   DATA[726,15] := 1.0;
   DATA[726,16] := 1.0;
   DATA[726,17] := 1.0;
   DATA[726,18] := 1.0;
   DATA[726,19] := 1.0;
   DATA[726,20] := 148.808;
   DATA[726,21] := 155.8318;
   DATA[726,22] := 1.720309;
   DATA[726,23] := 999.9744;
   DATA[726,24] := 2.0;
   DATA[726,25] := 2.0;
   DATA[726,26] := 7.878942;
   DATA[726,27] := 144.6039;
   DATA[726,28] := 263.1056;
   DATA[726,29] := 12.11228;
   DATA[726,30] := 1.734683;
   DATA[726,31] := 1.301652;
   DATA[726,32] := 0.7352687;
   DATA[726,33] := 0.3066329;
   DATA[726,34] := 2.0;
   DATA[726,35] := 251.474;
   DATA[726,36] := 1.730048;
   DATA[726,37] := 190.1275;
   DATA[726,38] := 0.000128152;
   DATA[726,39] := 1.0;
   DATA[727,0] := 2.455241;
   DATA[727,1] := 535.5254;
   DATA[727,2] := 2.0;
   DATA[727,3] := 2.0;
   DATA[727,4] := 262.1764;
   DATA[727,5] := 8.395475;
   DATA[727,6] := 327.6339;
   DATA[727,7] := 2.440393;
   DATA[727,8] := 2.0;
   DATA[727,9] := 2.0;
   DATA[727,10] := 2.0;
   DATA[727,11] := 1.987963;
   DATA[727,13] := 991.052;
   DATA[727,14] := 1.0;
   DATA[727,15] := 1.0;
   DATA[727,16] := 1.0;
   DATA[727,17] := 1.0;
   DATA[727,18] := 1.0;
   DATA[727,19] := 1.0;
   DATA[727,20] := 148.808;
   DATA[727,21] := 155.8318;
   DATA[727,22] := 1.720309;
   DATA[727,23] := 1000.051;
   DATA[727,24] := 2.0;
   DATA[727,25] := 2.0;
   DATA[727,26] := 7.878942;
   DATA[727,27] := 144.6039;
   DATA[727,28] := 263.1056;
   DATA[727,29] := 12.11228;
   DATA[727,30] := 1.734683;
   DATA[727,31] := 1.301652;
   DATA[727,32] := 0.7352687;
   DATA[727,33] := 0.3066329;
   DATA[727,34] := 2.0;
   DATA[727,35] := 251.474;
   DATA[727,36] := 1.730048;
   DATA[727,37] := 190.1275;
   DATA[727,38] := 0.000128152;
   DATA[727,39] := 1.0;
   DATA[728,0] := 2.444031;
   DATA[728,1] := 535.4076;
   DATA[728,2] := 2.0;
   DATA[728,3] := 2.0;
   DATA[728,4] := 262.1764;
   DATA[728,5] := 8.395475;
   DATA[728,6] := 327.6339;
   DATA[728,7] := 2.440393;
   DATA[728,8] := 2.0;
   DATA[728,9] := 2.0;
   DATA[728,10] := 2.0;
   DATA[728,11] := 1.987963;
   DATA[728,13] := 991.2122;
   DATA[728,14] := 1.0;
   DATA[728,15] := 1.0;
   DATA[728,16] := 1.0;
   DATA[728,17] := 1.0;
   DATA[728,18] := 1.0;
   DATA[728,19] := 1.0;
   DATA[728,20] := 148.808;
   DATA[728,21] := 155.8062;
   DATA[728,22] := 1.722231;
   DATA[728,23] := 999.8975;
   DATA[728,24] := 2.0;
   DATA[728,25] := 2.0;
   DATA[728,26] := 7.878942;
   DATA[728,27] := 144.5783;
   DATA[728,28] := 263.1056;
   DATA[728,29] := 12.11228;
   DATA[728,30] := 1.73212;
   DATA[728,31] := 1.292046;
   DATA[728,32] := 0.7352687;
   DATA[728,33] := 0.3066329;
   DATA[728,34] := 2.0;
   DATA[728,35] := 251.474;
   DATA[728,36] := 1.730048;
   DATA[728,37] := 190.1275;
   DATA[728,38] := 0.000128152;
   DATA[728,39] := 1.0;
   DATA[729,0] := 2.43026;
   DATA[729,1] := 535.3291;
   DATA[729,2] := 2.0;
   DATA[729,3] := 2.0;
   DATA[729,4] := 262.1764;
   DATA[729,5] := 8.395475;
   DATA[729,6] := 327.5827;
   DATA[729,7] := 2.440393;
   DATA[729,8] := 2.0;
   DATA[729,9] := 2.0;
   DATA[729,10] := 2.0;
   DATA[729,11] := 2.016774;
   DATA[729,13] := 991.5327;
   DATA[729,14] := 1.0;
   DATA[729,15] := 1.0;
   DATA[729,16] := 1.0;
   DATA[729,17] := 1.0;
   DATA[729,18] := 1.0;
   DATA[729,19] := 1.0;
   DATA[729,20] := 148.808;
   DATA[729,21] := 155.8062;
   DATA[729,22] := 1.722231;
   DATA[729,23] := 999.859;
   DATA[729,24] := 2.0;
   DATA[729,25] := 2.0;
   DATA[729,26] := 7.878942;
   DATA[729,27] := 144.5783;
   DATA[729,28] := 263.1056;
   DATA[729,29] := 12.11228;
   DATA[729,30] := 1.73212;
   DATA[729,31] := 1.292046;
   DATA[729,32] := 0.7352687;
   DATA[729,33] := 0.3066329;
   DATA[729,34] := 2.0;
   DATA[729,35] := 251.474;
   DATA[729,36] := 1.730048;
   DATA[729,37] := 190.1275;
   DATA[729,38] := 0.000128152;
   DATA[729,39] := 1.0;
   DATA[730,0] := 2.424815;
   DATA[730,1] := 535.4076;
   DATA[730,2] := 2.0;
   DATA[730,3] := 2.0;
   DATA[730,4] := 262.1764;
   DATA[730,5] := 8.395475;
   DATA[730,6] := 327.5827;
   DATA[730,7] := 2.440393;
   DATA[730,8] := 2.0;
   DATA[730,9] := 2.0;
   DATA[730,10] := 2.0;
   DATA[730,11] := 2.016774;
   DATA[730,13] := 991.6528;
   DATA[730,14] := 1.0;
   DATA[730,15] := 1.0;
   DATA[730,16] := 1.0;
   DATA[730,17] := 1.0;
   DATA[730,18] := 1.0;
   DATA[730,19] := 1.0;
   DATA[730,20] := 148.808;
   DATA[730,21] := 155.8062;
   DATA[730,22] := 1.722231;
   DATA[730,23] := 999.2822;
   DATA[730,24] := 2.0;
   DATA[730,25] := 2.0;
   DATA[730,26] := 7.878942;
   DATA[730,27] := 144.5783;
   DATA[730,28] := 263.1056;
   DATA[730,29] := 12.11228;
   DATA[730,30] := 1.73212;
   DATA[730,31] := 1.285513;
   DATA[730,32] := 0.7352687;
   DATA[730,33] := 0.3066329;
   DATA[730,34] := 2.0;
   DATA[730,35] := 251.474;
   DATA[730,36] := 1.730048;
   DATA[730,37] := 190.1275;
   DATA[730,38] := 0.000128152;
   DATA[730,39] := 1.0;
   DATA[731,0] := 2.424815;
   DATA[731,1] := 535.4861;
   DATA[731,2] := 2.0;
   DATA[731,3] := 2.0;
   DATA[731,4] := 262.1764;
   DATA[731,5] := 8.395475;
   DATA[731,6] := 327.5827;
   DATA[731,7] := 2.440393;
   DATA[731,8] := 2.0;
   DATA[731,9] := 2.0;
   DATA[731,10] := 2.0;
   DATA[731,11] := 2.016774;
   DATA[731,13] := 992.2136;
   DATA[731,14] := 1.0;
   DATA[731,15] := 1.0;
   DATA[731,16] := 1.0;
   DATA[731,17] := 1.0;
   DATA[731,18] := 1.0;
   DATA[731,19] := 1.0;
   DATA[731,20] := 148.808;
   DATA[731,21] := 155.8062;
   DATA[731,22] := 1.720053;
   DATA[731,23] := 999.2438;
   DATA[731,24] := 2.0;
   DATA[731,25] := 2.0;
   DATA[731,26] := 7.878942;
   DATA[731,27] := 144.5783;
   DATA[731,28] := 263.1056;
   DATA[731,29] := 12.11228;
   DATA[731,30] := 1.730838;
   DATA[731,31] := 1.274497;
   DATA[731,32] := 0.7352687;
   DATA[731,33] := 0.3066329;
   DATA[731,34] := 2.0;
   DATA[731,35] := 251.3939;
   DATA[731,36] := 1.730048;
   DATA[731,37] := 190.1275;
   DATA[731,38] := 0.000128152;
   DATA[731,39] := 1.0;
   DATA[732,0] := 2.452359;
   DATA[732,1] := 535.8002;
   DATA[732,2] := 2.0;
   DATA[732,3] := 2.0;
   DATA[732,4] := 262.1764;
   DATA[732,5] := 8.395475;
   DATA[732,6] := 327.5827;
   DATA[732,7] := 2.440393;
   DATA[732,8] := 2.0;
   DATA[732,9] := 2.0;
   DATA[732,10] := 2.0;
   DATA[732,11] := 2.016774;
   DATA[732,13] := 992.6942;
   DATA[732,14] := 1.0;
   DATA[732,15] := 1.0;
   DATA[732,16] := 1.0;
   DATA[732,17] := 1.0;
   DATA[732,18] := 1.0;
   DATA[732,19] := 1.0;
   DATA[732,20] := 148.808;
   DATA[732,21] := 155.8062;
   DATA[732,22] := 1.720053;
   DATA[732,23] := 998.4747;
   DATA[732,24] := 2.0;
   DATA[732,25] := 2.0;
   DATA[732,26] := 7.878942;
   DATA[732,27] := 144.5783;
   DATA[732,28] := 263.1056;
   DATA[732,29] := 12.11228;
   DATA[732,30] := 1.730838;
   DATA[732,31] := 1.280517;
   DATA[732,32] := 0.7352687;
   DATA[732,33] := 0.3066329;
   DATA[732,34] := 2.0;
   DATA[732,35] := 251.2977;
   DATA[732,36] := 1.730048;
   DATA[732,37] := 190.0154;
   DATA[732,38] := 0.000128152;
   DATA[732,39] := 1.0;
   DATA[733,0] := 2.48887;
   DATA[733,1] := 535.9179;
   DATA[733,2] := 2.0;
   DATA[733,3] := 2.0;
   DATA[733,4] := 262.1764;
   DATA[733,5] := 8.395475;
   DATA[733,6] := 327.5827;
   DATA[733,7] := 2.440393;
   DATA[733,8] := 2.0;
   DATA[733,9] := 2.0;
   DATA[733,10] := 2.0;
   DATA[733,11] := 2.010372;
   DATA[733,13] := 993.4552;
   DATA[733,14] := 1.0;
   DATA[733,15] := 1.0;
   DATA[733,16] := 1.0;
   DATA[733,17] := 1.0;
   DATA[733,18] := 1.0;
   DATA[733,19] := 1.0;
   DATA[733,20] := 148.808;
   DATA[733,21] := 155.8062;
   DATA[733,22] := 1.720053;
   DATA[733,23] := 998.6285;
   DATA[733,24] := 2.0;
   DATA[733,25] := 2.0;
   DATA[733,26] := 7.878942;
   DATA[733,27] := 144.5783;
   DATA[733,28] := 263.1056;
   DATA[733,29] := 12.11228;
   DATA[733,30] := 1.730838;
   DATA[733,31] := 1.28167;
   DATA[733,32] := 0.7352687;
   DATA[733,33] := 0.3066329;
   DATA[733,34] := 2.0;
   DATA[733,35] := 251.2977;
   DATA[733,36] := 1.730048;
   DATA[733,37] := 190.0154;
   DATA[733,38] := 0.000128152;
   DATA[733,39] := 1.0;
   DATA[734,0] := 2.532428;
   DATA[734,1] := 535.4076;
   DATA[734,2] := 2.0;
   DATA[734,3] := 2.0;
   DATA[734,4] := 262.1764;
   DATA[734,5] := 8.395475;
   DATA[734,6] := 327.5827;
   DATA[734,7] := 2.440393;
   DATA[734,8] := 2.0;
   DATA[734,9] := 2.0;
   DATA[734,10] := 2.0;
   DATA[734,11] := 2.003969;
   DATA[734,13] := 993.6956;
   DATA[734,14] := 1.0;
   DATA[734,15] := 1.0;
   DATA[734,16] := 1.0;
   DATA[734,17] := 1.0;
   DATA[734,18] := 1.0;
   DATA[734,19] := 1.0;
   DATA[734,20] := 148.808;
   DATA[734,21] := 155.8062;
   DATA[734,22] := 1.720053;
   DATA[734,23] := 998.1287;
   DATA[734,24] := 2.0;
   DATA[734,25] := 2.0;
   DATA[734,26] := 7.878942;
   DATA[734,27] := 144.7321;
   DATA[734,28] := 263.1056;
   DATA[734,29] := 12.11228;
   DATA[734,30] := 1.730838;
   DATA[734,31] := 1.296273;
   DATA[734,32] := 0.7352687;
   DATA[734,33] := 0.3066329;
   DATA[734,34] := 2.0;
   DATA[734,35] := 251.2977;
   DATA[734,36] := 1.730048;
   DATA[734,37] := 190.0154;
   DATA[734,38] := 0.000128152;
   DATA[734,39] := 1.0;
   DATA[735,0] := 2.572783;
   DATA[735,1] := 534.9366;
   DATA[735,2] := 2.0;
   DATA[735,3] := 2.0;
   DATA[735,4] := 262.1764;
   DATA[735,5] := 8.395475;
   DATA[735,6] := 327.5827;
   DATA[735,7] := 2.440393;
   DATA[735,8] := 2.0;
   DATA[735,9] := 2.0;
   DATA[735,10] := 2.0;
   DATA[735,11] := 2.003969;
   DATA[735,13] := 994.4165;
   DATA[735,14] := 1.0;
   DATA[735,15] := 1.0;
   DATA[735,16] := 1.0;
   DATA[735,17] := 1.0;
   DATA[735,18] := 1.0;
   DATA[735,19] := 1.0;
   DATA[735,20] := 148.808;
   DATA[735,21] := 155.8062;
   DATA[735,22] := 1.720053;
   DATA[735,23] := 998.244;
   DATA[735,24] := 2.0;
   DATA[735,25] := 2.0;
   DATA[735,26] := 7.878942;
   DATA[735,27] := 144.7321;
   DATA[735,28] := 263.1056;
   DATA[735,29] := 12.11228;
   DATA[735,30] := 1.730838;
   DATA[735,31] := 1.299475;
   DATA[735,32] := 0.7352687;
   DATA[735,33] := 0.3066329;
   DATA[735,34] := 2.0;
   DATA[735,35] := 251.2977;
   DATA[735,36] := 1.730048;
   DATA[735,37] := 189.9994;
   DATA[735,38] := 0.000128152;
   DATA[735,39] := 1.0;
   DATA[736,0] := 2.609615;
   DATA[736,1] := 534.8581;
   DATA[736,2] := 2.0;
   DATA[736,3] := 2.0;
   DATA[736,4] := 262.1764;
   DATA[736,5] := 8.395475;
   DATA[736,6] := 327.5827;
   DATA[736,7] := 2.440393;
   DATA[736,8] := 2.0;
   DATA[736,9] := 2.0;
   DATA[736,10] := 2.0;
   DATA[736,11] := 2.003969;
   DATA[736,13] := 994.8972;
   DATA[736,14] := 1.0;
   DATA[736,15] := 1.0;
   DATA[736,16] := 1.0;
   DATA[736,17] := 1.0;
   DATA[736,18] := 1.0;
   DATA[736,19] := 1.0;
   DATA[736,20] := 148.808;
   DATA[736,21] := 155.8062;
   DATA[736,22] := 1.720053;
   DATA[736,23] := 997.8979;
   DATA[736,24] := 2.0;
   DATA[736,25] := 2.0;
   DATA[736,26] := 7.878942;
   DATA[736,27] := 144.7321;
   DATA[736,28] := 263.1056;
   DATA[736,29] := 12.11228;
   DATA[736,30] := 1.730838;
   DATA[736,31] := 1.292046;
   DATA[736,32] := 0.7352687;
   DATA[736,33] := 0.3066329;
   DATA[736,34] := 2.0;
   DATA[736,35] := 251.2977;
   DATA[736,36] := 1.730048;
   DATA[736,37] := 189.9994;
   DATA[736,38] := 0.000128152;
   DATA[736,39] := 1.0;
   DATA[737,0] := 2.633635;
   DATA[737,1] := 534.5048;
   DATA[737,2] := 2.0;
   DATA[737,3] := 2.0;
   DATA[737,4] := 262.1764;
   DATA[737,5] := 8.395475;
   DATA[737,6] := 327.5827;
   DATA[737,7] := 2.440393;
   DATA[737,8] := 2.0;
   DATA[737,9] := 2.0;
   DATA[737,10] := 2.0;
   DATA[737,11] := 2.003969;
   DATA[737,13] := 995.4178;
   DATA[737,14] := 1.0;
   DATA[737,15] := 1.0;
   DATA[737,16] := 1.0;
   DATA[737,17] := 1.0;
   DATA[737,18] := 1.0;
   DATA[737,19] := 1.0;
   DATA[737,20] := 148.808;
   DATA[737,21] := 155.8062;
   DATA[737,22] := 1.720053;
   DATA[737,23] := 997.475;
   DATA[737,24] := 2.0;
   DATA[737,25] := 2.0;
   DATA[737,26] := 7.878942;
   DATA[737,27] := 144.7321;
   DATA[737,28] := 263.1056;
   DATA[737,29] := 12.11228;
   DATA[737,30] := 1.730838;
   DATA[737,31] := 1.28167;
   DATA[737,32] := 0.7352687;
   DATA[737,33] := 0.3066329;
   DATA[737,34] := 2.0;
   DATA[737,35] := 251.2977;
   DATA[737,36] := 1.730048;
   DATA[737,37] := 189.9994;
   DATA[737,38] := 0.000128152;
   DATA[737,39] := 1.0;
   DATA[738,0] := 2.649649;
   DATA[738,1] := 534.3085;
   DATA[738,2] := 2.0;
   DATA[738,3] := 2.0;
   DATA[738,4] := 262.1764;
   DATA[738,5] := 8.395475;
   DATA[738,6] := 327.5827;
   DATA[738,7] := 2.440393;
   DATA[738,8] := 2.0;
   DATA[738,9] := 2.0;
   DATA[738,10] := 2.0;
   DATA[738,11] := 2.003969;
   DATA[738,13] := 996.2991;
   DATA[738,14] := 1.0;
   DATA[738,15] := 1.0;
   DATA[738,16] := 1.0;
   DATA[738,17] := 1.0;
   DATA[738,18] := 1.0;
   DATA[738,19] := 1.0;
   DATA[738,20] := 148.808;
   DATA[738,21] := 155.8062;
   DATA[738,22] := 1.720053;
   DATA[738,23] := 996.9752;
   DATA[738,24] := 2.0;
   DATA[738,25] := 2.0;
   DATA[738,26] := 7.878942;
   DATA[738,27] := 144.7321;
   DATA[738,28] := 263.1056;
   DATA[738,29] := 12.11228;
   DATA[738,30] := 1.730838;
   DATA[738,31] := 1.28167;
   DATA[738,32] := 0.7352687;
   DATA[738,33] := 0.3066329;
   DATA[738,34] := 2.0;
   DATA[738,35] := 251.2977;
   DATA[738,36] := 1.730048;
   DATA[738,37] := 189.9994;
   DATA[738,38] := 0.000128152;
   DATA[738,39] := 1.0;
   DATA[739,0] := 2.653172;
   DATA[739,1] := 534.5048;
   DATA[739,2] := 2.0;
   DATA[739,3] := 2.0;
   DATA[739,4] := 262.1764;
   DATA[739,5] := 8.395475;
   DATA[739,6] := 327.5827;
   DATA[739,7] := 2.438984;
   DATA[739,8] := 2.0;
   DATA[739,9] := 2.0;
   DATA[739,10] := 2.0;
   DATA[739,11] := 2.013573;
   DATA[739,13] := 996.6595;
   DATA[739,14] := 1.0;
   DATA[739,15] := 1.0;
   DATA[739,16] := 1.0;
   DATA[739,17] := 1.0;
   DATA[739,18] := 1.0;
   DATA[739,19] := 1.0;
   DATA[739,20] := 148.808;
   DATA[739,21] := 155.8062;
   DATA[739,22] := 1.720053;
   DATA[739,23] := 996.5522;
   DATA[739,24] := 2.0;
   DATA[739,25] := 2.0;
   DATA[739,26] := 7.878942;
   DATA[739,27] := 144.7321;
   DATA[739,28] := 263.1056;
   DATA[739,29] := 12.11228;
   DATA[739,30] := 1.730838;
   DATA[739,31] := 1.272192;
   DATA[739,32] := 0.7352687;
   DATA[739,33] := 0.3066329;
   DATA[739,34] := 2.0;
   DATA[739,35] := 251.2977;
   DATA[739,36] := 1.730048;
   DATA[739,37] := 189.9994;
   DATA[739,38] := 0.000128152;
   DATA[739,39] := 1.0;
   DATA[740,0] := 2.6394;
   DATA[740,1] := 534.6618;
   DATA[740,2] := 2.0;
   DATA[740,3] := 2.0;
   DATA[740,4] := 262.1764;
   DATA[740,5] := 8.395475;
   DATA[740,6] := 327.5827;
   DATA[740,7] := 2.438984;
   DATA[740,8] := 2.0;
   DATA[740,9] := 2.0;
   DATA[740,10] := 2.0;
   DATA[740,11] := 2.016774;
   DATA[740,13] := 997.02;
   DATA[740,14] := 1.0;
   DATA[740,15] := 1.0;
   DATA[740,16] := 1.0;
   DATA[740,17] := 1.0;
   DATA[740,18] := 1.0;
   DATA[740,19] := 1.0;
   DATA[740,20] := 148.808;
   DATA[740,21] := 155.8062;
   DATA[740,22] := 1.720053;
   DATA[740,23] := 996.3984;
   DATA[740,24] := 2.0;
   DATA[740,25] := 2.0;
   DATA[740,26] := 7.878942;
   DATA[740,27] := 144.7321;
   DATA[740,28] := 263.1056;
   DATA[740,29] := 12.11228;
   DATA[740,30] := 1.733658;
   DATA[740,31] := 1.274497;
   DATA[740,32] := 0.7352687;
   DATA[740,33] := 0.3066329;
   DATA[740,34] := 2.0;
   DATA[740,35] := 251.2977;
   DATA[740,36] := 1.730048;
   DATA[740,37] := 189.9032;
   DATA[740,38] := 0.000128152;
   DATA[740,39] := 1.0;
   DATA[741,0] := 2.628191;
   DATA[741,1] := 534.9366;
   DATA[741,2] := 2.0;
   DATA[741,3] := 2.0;
   DATA[741,4] := 262.1764;
   DATA[741,5] := 8.395475;
   DATA[741,6] := 327.5827;
   DATA[741,7] := 2.438984;
   DATA[741,8] := 2.0;
   DATA[741,9] := 2.0;
   DATA[741,10] := 2.0;
   DATA[741,11] := 2.016774;
   DATA[741,13] := 997.8211;
   DATA[741,14] := 1.0;
   DATA[741,15] := 1.0;
   DATA[741,16] := 1.0;
   DATA[741,17] := 1.0;
   DATA[741,18] := 1.0;
   DATA[741,19] := 1.0;
   DATA[741,20] := 148.808;
   DATA[741,21] := 155.8062;
   DATA[741,22] := 1.717874;
   DATA[741,23] := 996.0139;
   DATA[741,24] := 2.0;
   DATA[741,25] := 2.0;
   DATA[741,26] := 7.878942;
   DATA[741,27] := 144.7321;
   DATA[741,28] := 263.1056;
   DATA[741,29] := 12.11228;
   DATA[741,30] := 1.733658;
   DATA[741,31] := 1.277828;
   DATA[741,32] := 0.7352687;
   DATA[741,33] := 0.3066329;
   DATA[741,34] := 2.0;
   DATA[741,35] := 251.2977;
   DATA[741,36] := 1.730048;
   DATA[741,37] := 189.9032;
   DATA[741,38] := 0.000128152;
   DATA[741,39] := 1.0;
   DATA[742,0] := 2.617942;
   DATA[742,1] := 535.0151;
   DATA[742,2] := 2.0;
   DATA[742,3] := 2.0;
   DATA[742,4] := 262.1764;
   DATA[742,5] := 8.395475;
   DATA[742,6] := 327.5827;
   DATA[742,7] := 2.438984;
   DATA[742,8] := 2.0;
   DATA[742,9] := 2.0;
   DATA[742,10] := 2.0;
   DATA[742,11] := 2.016774;
   DATA[742,13] := 998.462;
   DATA[742,14] := 1.0;
   DATA[742,15] := 1.0;
   DATA[742,16] := 1.0;
   DATA[742,17] := 1.0;
   DATA[742,18] := 1.0;
   DATA[742,19] := 1.0;
   DATA[742,20] := 148.808;
   DATA[742,21] := 155.8062;
   DATA[742,22] := 1.717874;
   DATA[742,23] := 995.6678;
   DATA[742,24] := 2.0;
   DATA[742,25] := 2.0;
   DATA[742,26] := 7.878942;
   DATA[742,27] := 144.7321;
   DATA[742,28] := 263.1056;
   DATA[742,29] := 12.11228;
   DATA[742,30] := 1.731095;
   DATA[742,31] := 1.271679;
   DATA[742,32] := 0.7352687;
   DATA[742,33] := 0.3066329;
   DATA[742,34] := 2.0;
   DATA[742,35] := 251.2977;
   DATA[742,36] := 1.730048;
   DATA[742,37] := 189.9032;
   DATA[742,38] := 0.000128152;
   DATA[742,39] := 1.0;
   DATA[743,0] := 2.617942;
   DATA[743,1] := 535.5254;
   DATA[743,2] := 2.0;
   DATA[743,3] := 2.0;
   DATA[743,4] := 262.1764;
   DATA[743,5] := 8.395475;
   DATA[743,6] := 327.5827;
   DATA[743,7] := 2.438984;
   DATA[743,8] := 2.0;
   DATA[743,9] := 2.0;
   DATA[743,10] := 2.0;
   DATA[743,11] := 2.016774;
   DATA[743,13] := 999.5434;
   DATA[743,14] := 1.0;
   DATA[743,15] := 1.0;
   DATA[743,16] := 1.0;
   DATA[743,17] := 1.0;
   DATA[743,18] := 1.0;
   DATA[743,19] := 1.0;
   DATA[743,20] := 148.808;
   DATA[743,21] := 155.8062;
   DATA[743,22] := 1.717874;
   DATA[743,23] := 995.091;
   DATA[743,24] := 2.0;
   DATA[743,25] := 2.0;
   DATA[743,26] := 7.878942;
   DATA[743,27] := 144.7321;
   DATA[743,28] := 263.1056;
   DATA[743,29] := 12.11228;
   DATA[743,30] := 1.731095;
   DATA[743,31] := 1.274625;
   DATA[743,32] := 0.7352687;
   DATA[743,33] := 0.3066329;
   DATA[743,34] := 2.0;
   DATA[743,35] := 251.2977;
   DATA[743,36] := 1.730048;
   DATA[743,37] := 189.9032;
   DATA[743,38] := 0.000128152;
   DATA[743,39] := 1.0;
   DATA[744,0] := 2.601928;
   DATA[744,1] := 536.2319;
   DATA[744,2] := 2.0;
   DATA[744,3] := 1.0;
   DATA[744,4] := 262.1764;
   DATA[744,5] := 8.395475;
   DATA[744,6] := 327.5827;
   DATA[744,7] := 2.438984;
   DATA[744,8] := 2.0;
   DATA[744,9] := 2.0;
   DATA[744,10] := 2.0;
   DATA[744,11] := 2.016774;
   DATA[744,13] := 1000.144;
   DATA[744,14] := 1.0;
   DATA[744,15] := 1.0;
   DATA[744,16] := 1.0;
   DATA[744,17] := 1.0;
   DATA[744,18] := 1.0;
   DATA[744,19] := 1.0;
   DATA[744,20] := 148.808;
   DATA[744,21] := 155.8062;
   DATA[744,22] := 1.717874;
   DATA[744,23] := 994.7065;
   DATA[744,24] := 2.0;
   DATA[744,25] := 2.0;
   DATA[744,26] := 7.878942;
   DATA[744,27] := 144.7321;
   DATA[744,28] := 263.1056;
   DATA[744,29] := 12.11228;
   DATA[744,30] := 1.731095;
   DATA[744,31] := 1.277059;
   DATA[744,32] := 0.7352687;
   DATA[744,33] := 0.3066329;
   DATA[744,34] := 2.0;
   DATA[744,35] := 251.2977;
   DATA[744,36] := 1.730048;
   DATA[744,37] := 189.9032;
   DATA[744,38] := 0.000128152;
   DATA[744,39] := 1.0;
   DATA[745,0] := 2.591359;
   DATA[745,1] := 537.0562;
   DATA[745,2] := 2.0;
   DATA[745,3] := 1.0;
   DATA[745,4] := 262.1764;
   DATA[745,5] := 8.395475;
   DATA[745,6] := 327.5827;
   DATA[745,7] := 2.438984;
   DATA[745,9] := 1.0;
   DATA[745,10] := 1.0;
   DATA[745,11] := 2.016774;
   DATA[745,13] := 1001.025;
   DATA[745,14] := 1.0;
   DATA[745,15] := 1.0;
   DATA[745,16] := 1.0;
   DATA[745,17] := 1.0;
   DATA[745,18] := 1.0;
   DATA[745,19] := 1.0;
   DATA[745,20] := 148.808;
   DATA[745,21] := 155.8062;
   DATA[745,22] := 1.717874;
   DATA[745,23] := 994.1297;
   DATA[745,24] := 2.0;
   DATA[745,25] := 2.0;
   DATA[745,26] := 7.878942;
   DATA[745,27] := 144.7321;
   DATA[745,28] := 263.1056;
   DATA[745,29] := 12.11228;
   DATA[745,30] := 1.731095;
   DATA[745,31] := 1.275394;
   DATA[745,32] := 0.7352687;
   DATA[745,33] := 0.3066329;
   DATA[745,34] := 2.0;
   DATA[745,35] := 251.2977;
   DATA[745,36] := 1.730048;
   DATA[745,37] := 189.9032;
   DATA[745,38] := 0.000128152;
   DATA[745,39] := 1.0;
   DATA[746,0] := 2.567338;
   DATA[746,1] := 537.4488;
   DATA[746,2] := 2.0;
   DATA[746,3] := 1.0;
   DATA[746,4] := 262.1764;
   DATA[746,5] := 8.395475;
   DATA[746,6] := 327.5827;
   DATA[746,7] := 2.42886;
   DATA[746,9] := 1.0;
   DATA[746,10] := 1.0;
   DATA[746,11] := 2.016774;
   DATA[746,13] := 1001.706;
   DATA[746,14] := 1.0;
   DATA[746,15] := 1.0;
   DATA[746,16] := 1.0;
   DATA[746,17] := 1.0;
   DATA[746,18] := 1.0;
   DATA[746,19] := 1.0;
   DATA[746,20] := 148.808;
   DATA[746,21] := 155.8062;
   DATA[746,22] := 1.71813;
   DATA[746,23] := 994.0143;
   DATA[746,24] := 2.0;
   DATA[746,25] := 2.0;
   DATA[746,26] := 7.878942;
   DATA[746,27] := 144.7321;
   DATA[746,28] := 263.1056;
   DATA[746,29] := 12.11228;
   DATA[746,30] := 1.731095;
   DATA[746,31] := 1.281542;
   DATA[746,32] := 0.7352687;
   DATA[746,33] := 0.3066329;
   DATA[746,34] := 2.0;
   DATA[746,35] := 251.2977;
   DATA[746,36] := 1.730048;
   DATA[746,37] := 189.9032;
   DATA[746,38] := 0.000128152;
   DATA[746,39] := 1.0;
   DATA[747,0] := 2.556449;
   DATA[747,1] := 537.959;
   DATA[747,2] := 2.0;
   DATA[747,3] := 1.0;
   DATA[747,4] := 262.1764;
   DATA[747,5] := 8.395475;
   DATA[747,6] := 327.5827;
   DATA[747,7] := 2.323647;
   DATA[747,9] := 1.0;
   DATA[747,10] := 1.0;
   DATA[747,11] := 2.016774;
   DATA[747,13] := 1002.908;
   DATA[747,14] := 1.0;
   DATA[747,15] := 1.0;
   DATA[747,16] := 1.0;
   DATA[747,17] := 1.0;
   DATA[747,18] := 1.0;
   DATA[747,19] := 1.0;
   DATA[747,20] := 148.808;
   DATA[747,21] := 155.8062;
   DATA[747,22] := 1.720309;
   DATA[747,23] := 993.899;
   DATA[747,24] := 2.0;
   DATA[747,25] := 2.0;
   DATA[747,26] := 7.878942;
   DATA[747,27] := 144.7321;
   DATA[747,28] := 263.1056;
   DATA[747,29] := 12.11228;
   DATA[747,30] := 1.731095;
   DATA[747,31] := 1.291789;
   DATA[747,32] := 0.7352687;
   DATA[747,33] := 0.3066329;
   DATA[747,34] := 2.0;
   DATA[747,35] := 251.2977;
   DATA[747,36] := 1.730048;
   DATA[747,37] := 190.0154;
   DATA[747,38] := 0.000128152;
   DATA[747,39] := 1.0;
   DATA[748,0] := 2.536912;
   DATA[748,1] := 538.1553;
   DATA[748,2] := 2.0;
   DATA[748,3] := 1.0;
   DATA[748,4] := 262.1764;
   DATA[748,5] := 8.399321;
   DATA[748,6] := 327.5827;
   DATA[748,7] := 2.09464;
   DATA[748,9] := 1.0;
   DATA[748,10] := 1.0;
   DATA[748,11] := 2.010372;
   DATA[748,13] := 1003.228;
   DATA[748,14] := 1.0;
   DATA[748,15] := 1.0;
   DATA[748,16] := 1.0;
   DATA[748,17] := 1.0;
   DATA[748,18] := 1.0;
   DATA[748,19] := 1.0;
   DATA[748,20] := 148.808;
   DATA[748,21] := 155.8062;
   DATA[748,22] := 1.72159;
   DATA[748,23] := 993.8221;
   DATA[748,24] := 2.0;
   DATA[748,25] := 2.0;
   DATA[748,26] := 7.878942;
   DATA[748,27] := 144.7321;
   DATA[748,28] := 263.1056;
   DATA[748,29] := 12.11228;
   DATA[748,30] := 1.731095;
   DATA[748,31] := 1.288971;
   DATA[748,32] := 0.7352687;
   DATA[748,33] := 0.3066329;
   DATA[748,34] := 2.0;
   DATA[748,35] := 251.2977;
   DATA[748,36] := 1.730048;
   DATA[748,37] := 190.0795;
   DATA[748,38] := 0.000128152;
   DATA[748,39] := 1.0;
   DATA[749,0] := 2.514813;
   DATA[749,1] := 538.5479;
   DATA[749,2] := 2.0;
   DATA[749,3] := 1.0;
   DATA[749,4] := 262.1764;
   DATA[749,5] := 8.399321;
   DATA[749,6] := 327.5827;
   DATA[749,7] := 1.782847;
   DATA[749,9] := 1.0;
   DATA[749,10] := 1.0;
   DATA[749,11] := 2.010372;
   DATA[749,13] := 1003.749;
   DATA[749,14] := 1.0;
   DATA[749,15] := 1.0;
   DATA[749,16] := 1.0;
   DATA[749,17] := 1.0;
   DATA[749,18] := 1.0;
   DATA[749,19] := 1.0;
   DATA[749,20] := 148.808;
   DATA[749,21] := 155.6524;
   DATA[749,22] := 1.721975;
   DATA[749,23] := 993.4376;
   DATA[749,24] := 2.0;
   DATA[749,25] := 2.0;
   DATA[749,26] := 7.878942;
   DATA[749,27] := 144.7321;
   DATA[749,28] := 263.1056;
   DATA[749,29] := 12.11228;
   DATA[749,30] := 1.731095;
   DATA[749,31] := 1.282951;
   DATA[749,32] := 0.7352687;
   DATA[749,33] := 0.3066329;
   DATA[749,34] := 2.0;
   DATA[749,35] := 251.2977;
   DATA[749,36] := 1.730048;
   DATA[749,37] := 190.0795;
   DATA[749,38] := 0.000128152;
   DATA[749,39] := 1.0;
   DATA[750,0] := 2.496237;
   DATA[750,1] := 538.8619;
   DATA[750,2] := 2.0;
   DATA[750,3] := 1.0;
   DATA[750,4] := 262.1764;
   DATA[750,5] := 8.399321;
   DATA[750,6] := 327.5827;
   DATA[750,7] := 1.39365;
   DATA[750,9] := 1.0;
   DATA[750,10] := 1.0;
   DATA[750,11] := 2.010372;
   DATA[750,13] := 1004.31;
   DATA[750,14] := 1.0;
   DATA[750,15] := 1.0;
   DATA[750,16] := 1.0;
   DATA[750,17] := 1.0;
   DATA[750,18] := 1.0;
   DATA[750,19] := 1.0;
   DATA[750,20] := 148.808;
   DATA[750,21] := 155.6524;
   DATA[750,22] := 1.72159;
   DATA[750,23] := 993.6683;
   DATA[750,24] := 2.0;
   DATA[750,25] := 2.0;
   DATA[750,26] := 7.878942;
   DATA[750,27] := 144.7321;
   DATA[750,28] := 263.1056;
   DATA[750,29] := 12.11228;
   DATA[750,30] := 1.731095;
   DATA[750,31] := 1.282439;
   DATA[750,32] := 0.7352687;
   DATA[750,33] := 0.3066329;
   DATA[750,34] := 2.0;
   DATA[750,35] := 251.2977;
   DATA[750,36] := 1.730048;
   DATA[750,37] := 190.0795;
   DATA[750,38] := 0.000128152;
   DATA[750,39] := 1.0;
   DATA[751,0] := 2.480223;
   DATA[751,1] := 538.8226;
   DATA[751,2] := 2.0;
   DATA[751,3] := 1.0;
   DATA[751,4] := 262.1764;
   DATA[751,5] := 8.399321;
   DATA[751,6] := 327.5827;
   DATA[751,7] := 1.022395;
   DATA[751,9] := 1.0;
   DATA[751,10] := 1.0;
   DATA[751,11] := 2.010372;
   DATA[751,13] := 1004.951;
   DATA[751,14] := 1.0;
   DATA[751,15] := 1.0;
   DATA[751,16] := 1.0;
   DATA[751,17] := 1.0;
   DATA[751,18] := 1.0;
   DATA[751,19] := 1.0;
   DATA[751,20] := 148.808;
   DATA[751,21] := 155.6524;
   DATA[751,22] := 1.719668;
   DATA[751,23] := 993.1684;
   DATA[751,24] := 2.0;
   DATA[751,25] := 2.0;
   DATA[751,26] := 7.878942;
   DATA[751,27] := 144.7321;
   DATA[751,28] := 263.1056;
   DATA[751,29] := 12.11228;
   DATA[751,30] := 1.731735;
   DATA[751,31] := 1.281927;
   DATA[751,32] := 0.7352687;
   DATA[751,33] := 0.3066329;
   DATA[751,34] := 2.0;
   DATA[751,35] := 251.2977;
   DATA[751,36] := 1.762086;
   DATA[751,37] := 190.0795;
   DATA[751,38] := 0.000128152;
   DATA[751,39] := 1.0;
   DATA[752,0] := 2.464849;
   DATA[752,1] := 538.9796;
   DATA[752,2] := 2.0;
   DATA[752,3] := 1.0;
   DATA[752,4] := 262.1764;
   DATA[752,5] := 8.399321;
   DATA[752,6] := 327.3263;
   DATA[752,7] := 0.6416557;
   DATA[752,9] := 1.0;
   DATA[752,10] := 1.0;
   DATA[752,11] := 2.010372;
   DATA[752,13] := 1005.351;
   DATA[752,14] := 1.0;
   DATA[752,15] := 1.0;
   DATA[752,16] := 1.0;
   DATA[752,17] := 1.0;
   DATA[752,18] := 1.0;
   DATA[752,19] := 1.0;
   DATA[752,20] := 148.808;
   DATA[752,21] := 155.6524;
   DATA[752,22] := 1.719668;
   DATA[752,23] := 993.1299;
   DATA[752,24] := 2.0;
   DATA[752,25] := 2.0;
   DATA[752,26] := 7.878942;
   DATA[752,27] := 144.7321;
   DATA[752,28] := 263.1056;
   DATA[752,29] := 12.11228;
   DATA[752,30] := 1.734427;
   DATA[752,31] := 1.288075;
   DATA[752,32] := 0.7352687;
   DATA[752,33] := 0.3066329;
   DATA[752,34] := 2.0;
   DATA[752,35] := 251.2977;
   DATA[752,36] := 1.762086;
   DATA[752,37] := 190.0795;
   DATA[752,38] := 0.000128152;
   DATA[752,39] := 1.0;
   DATA[753,0] := 2.449156;
   DATA[753,1] := 539.1759;
   DATA[753,2] := 2.0;
   DATA[753,3] := 1.0;
   DATA[753,4] := 262.1764;
   DATA[753,5] := 8.399321;
   DATA[753,6] := 326.9931;
   DATA[753,7] := 0.3813795;
   DATA[753,8] := 1.0;
   DATA[753,9] := 1.0;
   DATA[753,10] := 1.0;
   DATA[753,11] := 2.010372;
   DATA[753,13] := 1006.272;
   DATA[753,14] := 1.0;
   DATA[753,15] := 1.0;
   DATA[753,16] := 1.0;
   DATA[753,17] := 1.0;
   DATA[753,18] := 1.0;
   DATA[753,19] := 1.0;
   DATA[753,20] := 148.808;
   DATA[753,21] := 155.6524;
   DATA[753,22] := 1.721719;
   DATA[753,23] := 992.361;
   DATA[753,24] := 2.0;
   DATA[753,25] := 2.0;
   DATA[753,26] := 7.878942;
   DATA[753,27] := 144.7321;
   DATA[753,28] := 263.1056;
   DATA[753,29] := 12.11228;
   DATA[753,30] := 1.734427;
   DATA[753,31] := 1.291277;
   DATA[753,32] := 0.7352687;
   DATA[753,33] := 0.3066329;
   DATA[753,34] := 2.0;
   DATA[753,35] := 251.2977;
   DATA[753,36] := 1.762086;
   DATA[753,37] := 190.0795;
   DATA[753,38] := 0.000128152;
   DATA[753,39] := 1.0;
   DATA[754,0] := 2.433462;
   DATA[754,1] := 539.7646;
   DATA[754,2] := 2.0;
   DATA[754,3] := 1.0;
   DATA[754,4] := 262.1764;
   DATA[754,5] := 8.399321;
   DATA[754,6] := 326.7111;
   DATA[754,7] := 0.2296479;
   DATA[754,8] := 1.0;
   DATA[754,9] := 1.0;
   DATA[754,10] := 1.0;
   DATA[754,11] := 2.010372;
   DATA[754,13] := 1006.753;
   DATA[754,14] := 1.0;
   DATA[754,15] := 1.0;
   DATA[754,16] := 1.0;
   DATA[754,17] := 1.0;
   DATA[754,18] := 1.0;
   DATA[754,19] := 1.0;
   DATA[754,20] := 148.808;
   DATA[754,21] := 155.4473;
   DATA[754,22] := 1.721719;
   DATA[754,23] := 992.3225;
   DATA[754,24] := 2.0;
   DATA[754,25] := 2.0;
   DATA[754,26] := 7.878942;
   DATA[754,27] := 144.7321;
   DATA[754,28] := 263.1056;
   DATA[754,29] := 12.11228;
   DATA[754,30] := 1.734427;
   DATA[754,31] := 1.291405;
   DATA[754,32] := 0.7352687;
   DATA[754,33] := 0.3066329;
   DATA[754,34] := 2.0;
   DATA[754,35] := 251.2977;
   DATA[754,36] := 1.762086;
   DATA[754,37] := 190.0795;
   DATA[754,38] := 0.000128152;
   DATA[754,39] := 1.0;
   DATA[755,0] := 2.423213;
   DATA[755,1] := 539.804;
   DATA[755,2] := 2.0;
   DATA[755,3] := 1.0;
   DATA[755,4] := 262.1764;
   DATA[755,5] := 8.399321;
   DATA[755,6] := 326.7111;
   DATA[755,7] := 0.1289206;
   DATA[755,8] := 1.0;
   DATA[755,9] := 1.0;
   DATA[755,10] := 1.0;
   DATA[755,11] := 2.010372;
   DATA[755,13] := 1006.953;
   DATA[755,14] := 1.0;
   DATA[755,15] := 1.0;
   DATA[755,16] := 1.0;
   DATA[755,17] := 1.0;
   DATA[755,18] := 1.0;
   DATA[755,19] := 1.0;
   DATA[755,20] := 148.808;
   DATA[755,21] := 155.4217;
   DATA[755,22] := 1.721719;
   DATA[755,23] := 991.5535;
   DATA[755,24] := 2.0;
   DATA[755,25] := 2.0;
   DATA[755,26] := 7.878942;
   DATA[755,27] := 144.8603;
   DATA[755,28] := 263.1056;
   DATA[755,29] := 12.11228;
   DATA[755,30] := 1.733786;
   DATA[755,31] := 1.291405;
   DATA[755,32] := 0.7352687;
   DATA[755,33] := 0.3066329;
   DATA[755,34] := 2.0;
   DATA[755,35] := 251.2977;
   DATA[755,36] := 1.762086;
   DATA[755,37] := 190.0154;
   DATA[755,38] := 0.000128152;
   DATA[755,39] := 1.0;
   DATA[756,0] := 2.41905;
   DATA[756,1] := 540.3535;
   DATA[756,2] := 2.0;
   DATA[756,3] := 1.0;
   DATA[756,4] := 262.1764;
   DATA[756,5] := 8.399321;
   DATA[756,6] := 326.5573;
   DATA[756,7] := 0.070099;
   DATA[756,8] := 1.0;
   DATA[756,9] := 1.0;
   DATA[756,10] := 1.0;
   DATA[756,11] := 2.010372;
   DATA[756,13] := 1007.474;
   DATA[756,14] := 1.0;
   DATA[756,15] := 1.0;
   DATA[756,16] := 1.0;
   DATA[756,17] := 1.0;
   DATA[756,18] := 1.0;
   DATA[756,19] := 1.0;
   DATA[756,20] := 148.808;
   DATA[756,21] := 155.4217;
   DATA[756,22] := 1.720053;
   DATA[756,23] := 991.7457;
   DATA[756,24] := 2.0;
   DATA[756,25] := 2.0;
   DATA[756,26] := 7.878942;
   DATA[756,27] := 144.8603;
   DATA[756,28] := 263.1056;
   DATA[756,29] := 12.11228;
   DATA[756,30] := 1.731223;
   DATA[756,31] := 1.29243;
   DATA[756,32] := 0.7352687;
   DATA[756,33] := 0.3066329;
   DATA[756,34] := 2.0;
   DATA[756,35] := 251.2977;
   DATA[756,36] := 1.762086;
   DATA[756,37] := 189.8872;
   DATA[756,38] := 0.000128152;
   DATA[756,39] := 1.0;
   DATA[757,0] := 2.41905;
   DATA[757,1] := 540.5497;
   DATA[757,2] := 2.0;
   DATA[757,3] := 1.0;
   DATA[757,4] := 262.1764;
   DATA[757,5] := 8.401243;
   DATA[757,6] := 325.9677;
   DATA[757,7] := 0.03575433;
   DATA[757,8] := 1.0;
   DATA[757,9] := 1.0;
   DATA[757,10] := 1.0;
   DATA[757,11] := 2.010372;
   DATA[757,13] := 1007.835;
   DATA[757,14] := 1.0;
   DATA[757,15] := 1.0;
   DATA[757,16] := 1.0;
   DATA[757,17] := 1.0;
   DATA[757,18] := 1.0;
   DATA[757,19] := 1.0;
   DATA[757,20] := 148.808;
   DATA[757,21] := 155.4217;
   DATA[757,22] := 1.719668;
   DATA[757,23] := 991.3997;
   DATA[757,24] := 2.0;
   DATA[757,25] := 2.0;
   DATA[757,26] := 7.878942;
   DATA[757,27] := 144.8603;
   DATA[757,28] := 263.1056;
   DATA[757,29] := 12.11228;
   DATA[757,30] := 1.731223;
   DATA[757,31] := 1.302165;
   DATA[757,32] := 0.7352687;
   DATA[757,33] := 0.3066329;
   DATA[757,34] := 2.0;
   DATA[757,35] := 251.1535;
   DATA[757,36] := 1.762086;
   DATA[757,37] := 189.8552;
   DATA[757,38] := 0.000128152;
   DATA[757,39] := 1.0;
   DATA[758,0] := 2.437626;
   DATA[758,1] := 541.0992;
   DATA[758,2] := 2.0;
   DATA[758,3] := 1.0;
   DATA[758,4] := 262.1764;
   DATA[758,5] := 8.401243;
   DATA[758,6] := 325.4294;
   DATA[758,7] := 0.01435299;
   DATA[758,8] := 1.0;
   DATA[758,9] := 1.0;
   DATA[758,10] := 1.0;
   DATA[758,11] := 2.010372;
   DATA[758,13] := 1008.355;
   DATA[758,14] := 1.0;
   DATA[758,15] := 1.0;
   DATA[758,16] := 1.0;
   DATA[758,17] := 1.0;
   DATA[758,18] := 1.0;
   DATA[758,19] := 1.0;
   DATA[758,20] := 148.808;
   DATA[758,21] := 155.4217;
   DATA[758,22] := 1.719668;
   DATA[758,23] := 991.3228;
   DATA[758,24] := 2.0;
   DATA[758,25] := 2.0;
   DATA[758,26] := 7.878942;
   DATA[758,27] := 144.8603;
   DATA[758,28] := 263.1056;
   DATA[758,29] := 12.11228;
   DATA[758,30] := 1.731223;
   DATA[758,31] := 1.311387;
   DATA[758,32] := 0.7352687;
   DATA[758,33] := 0.3066329;
   DATA[758,34] := 2.0;
   DATA[758,35] := 251.1055;
   DATA[758,36] := 1.762086;
   DATA[758,37] := 189.8552;
   DATA[758,38] := 0.000128152;
   DATA[758,39] := 1.0;
   DATA[759,0] := 2.461006;
   DATA[759,1] := 540.8245;
   DATA[759,2] := 2.0;
   DATA[759,3] := 1.0;
   DATA[759,4] := 262.1764;
   DATA[759,5] := 8.405088;
   DATA[759,6] := 325.4294;
   DATA[759,7] := 0.000512607;
   DATA[759,8] := 1.0;
   DATA[759,9] := 1.0;
   DATA[759,10] := 1.0;
   DATA[759,11] := 2.010372;
   DATA[759,13] := 1008.275;
   DATA[759,14] := 1.0;
   DATA[759,15] := 1.0;
   DATA[759,16] := 1.0;
   DATA[759,17] := 1.0;
   DATA[759,18] := 1.0;
   DATA[759,19] := 1.0;
   DATA[759,20] := 148.808;
   DATA[759,21] := 155.5242;
   DATA[759,22] := 1.719668;
   DATA[759,23] := 990.4768;
   DATA[759,24] := 2.0;
   DATA[759,25] := 2.0;
   DATA[759,26] := 7.878942;
   DATA[759,27] := 144.8603;
   DATA[759,28] := 263.1056;
   DATA[759,29] := 12.11228;
   DATA[759,30] := 1.731223;
   DATA[759,31] := 1.306648;
   DATA[759,32] := 0.7352687;
   DATA[759,33] := 0.3066329;
   DATA[759,34] := 2.0;
   DATA[759,35] := 251.0734;
   DATA[759,36] := 1.746067;
   DATA[759,37] := 189.8231;
   DATA[759,38] := 0.000128152;
   DATA[759,39] := 1.0;
   DATA[760,0] := 2.478621;
   DATA[760,1] := 541.4918;
   DATA[760,2] := 2.0;
   DATA[760,3] := 1.0;
   DATA[760,4] := 262.1764;
   DATA[760,5] := 8.40605;
   DATA[760,6] := 324.7885;
   DATA[760,7] := 0.000512607;
   DATA[760,8] := 1.0;
   DATA[760,9] := 1.0;
   DATA[760,10] := 1.0;
   DATA[760,11] := 2.010372;
   DATA[760,13] := 1008.355;
   DATA[760,14] := 1.0;
   DATA[760,15] := 1.0;
   DATA[760,16] := 1.0;
   DATA[760,17] := 1.0;
   DATA[760,18] := 1.0;
   DATA[760,19] := 1.0;
   DATA[760,20] := 148.808;
   DATA[760,21] := 155.5242;
   DATA[760,22] := 1.719924;
   DATA[760,23] := 990.3999;
   DATA[760,24] := 2.0;
   DATA[760,25] := 2.0;
   DATA[760,26] := 7.878942;
   DATA[760,27] := 144.8603;
   DATA[760,28] := 263.1056;
   DATA[760,29] := 11.95847;
   DATA[760,30] := 1.731223;
   DATA[760,31] := 1.308185;
   DATA[760,32] := 0.7352687;
   DATA[760,33] := 0.3066329;
   DATA[760,34] := 2.0;
   DATA[760,35] := 250.8652;
   DATA[760,36] := 1.746067;
   DATA[760,37] := 189.727;
   DATA[760,38] := 0.000128152;
   DATA[760,39] := 1.0;
   DATA[761,0] := 2.502642;
   DATA[761,1] := 542.0021;
   DATA[761,2] := 2.0;
   DATA[761,3] := 1.0;
   DATA[761,4] := 262.1764;
   DATA[761,5] := 8.40605;
   DATA[761,6] := 324.1989;
   DATA[761,7] := 0.000512607;
   DATA[761,8] := 1.0;
   DATA[761,9] := 1.0;
   DATA[761,10] := 1.0;
   DATA[761,11] := 2.010372;
   DATA[761,13] := 1008.636;
   DATA[761,14] := 1.0;
   DATA[761,15] := 1.0;
   DATA[761,16] := 1.0;
   DATA[761,17] := 1.0;
   DATA[761,18] := 1.0;
   DATA[761,19] := 1.0;
   DATA[761,20] := 148.808;
   DATA[761,21] := 155.5242;
   DATA[761,22] := 1.719924;
   DATA[761,23] := 990.0154;
   DATA[761,24] := 2.0;
   DATA[761,25] := 2.0;
   DATA[761,26] := 7.878942;
   DATA[761,27] := 144.8603;
   DATA[761,28] := 263.1056;
   DATA[761,29] := 11.95847;
   DATA[761,30] := 1.731223;
   DATA[761,31] := 1.3119;
   DATA[761,32] := 0.7352687;
   DATA[761,33] := 0.3066329;
   DATA[761,34] := 2.0;
   DATA[761,35] := 250.8652;
   DATA[761,36] := 1.746067;
   DATA[761,37] := 189.727;
   DATA[761,38] := 0.000128152;
   DATA[761,39] := 1.0;
   DATA[762,0] := 2.515453;
   DATA[762,1] := 542.3553;
   DATA[762,2] := 2.0;
   DATA[762,3] := 1.0;
   DATA[762,4] := 262.1764;
   DATA[762,5] := 8.408293;
   DATA[762,6] := 323.7375;
   DATA[762,7] := 0.000512607;
   DATA[762,8] := 1.0;
   DATA[762,9] := 1.0;
   DATA[762,10] := 1.0;
   DATA[762,11] := 2.035982;
   DATA[762,13] := 1008.475;
   DATA[762,14] := 1.0;
   DATA[762,15] := 1.0;
   DATA[762,16] := 1.0;
   DATA[762,17] := 1.0;
   DATA[762,18] := 1.0;
   DATA[762,19] := 1.0;
   DATA[762,20] := 148.808;
   DATA[762,21] := 155.5242;
   DATA[762,22] := 1.719924;
   DATA[762,23] := 989.8231;
   DATA[762,24] := 2.0;
   DATA[762,25] := 2.0;
   DATA[762,26] := 7.878942;
   DATA[762,27] := 144.8603;
   DATA[762,28] := 263.1056;
   DATA[762,29] := 11.95847;
   DATA[762,30] := 1.731223;
   DATA[762,31] := 1.304855;
   DATA[762,32] := 0.7352687;
   DATA[762,33] := 0.3066329;
   DATA[762,34] := 2.0;
   DATA[762,35] := 250.8652;
   DATA[762,36] := 1.746067;
   DATA[762,37] := 189.6629;
   DATA[762,38] := 0.000128152;
   DATA[762,39] := 1.0;
   DATA[763,0] := 2.528264;
   DATA[763,1] := 542.9442;
   DATA[763,2] := 2.0;
   DATA[763,3] := 1.0;
   DATA[763,4] := 262.1764;
   DATA[763,5] := 8.412458;
   DATA[763,6] := 323.3017;
   DATA[763,7] := 0.000512607;
   DATA[763,8] := 1.0;
   DATA[763,9] := 1.0;
   DATA[763,10] := 1.0;
   DATA[763,11] := 2.035982;
   DATA[763,13] := 1008.876;
   DATA[763,14] := 1.0;
   DATA[763,15] := 1.0;
   DATA[763,16] := 1.0;
   DATA[763,17] := 1.0;
   DATA[763,18] := 1.0;
   DATA[763,19] := 1.0;
   DATA[763,20] := 148.808;
   DATA[763,21] := 155.5242;
   DATA[763,22] := 1.719924;
   DATA[763,23] := 989.5155;
   DATA[763,24] := 2.0;
   DATA[763,25] := 2.0;
   DATA[763,26] := 7.878942;
   DATA[763,27] := 144.8603;
   DATA[763,28] := 263.1056;
   DATA[763,29] := 11.95847;
   DATA[763,30] := 1.731095;
   DATA[763,31] := 1.291789;
   DATA[763,32] := 0.7352687;
   DATA[763,33] := 0.3066329;
   DATA[763,34] := 2.0;
   DATA[763,35] := 250.8652;
   DATA[763,36] := 1.537821;
   DATA[763,37] := 189.6629;
   DATA[763,38] := 0.000128152;
   DATA[763,39] := 1.0;
   DATA[764,0] := 2.533068;
   DATA[764,1] := 543.4937;
   DATA[764,2] := 2.0;
   DATA[764,3] := 1.0;
   DATA[764,4] := 262.1764;
   DATA[764,5] := 8.412458;
   DATA[764,6] := 323.0197;
   DATA[764,7] := 0.000512607;
   DATA[764,8] := 1.0;
   DATA[764,9] := 1.0;
   DATA[764,10] := 1.0;
   DATA[764,11] := 2.026378;
   DATA[764,13] := 1008.836;
   DATA[764,14] := 1.0;
   DATA[764,15] := 1.0;
   DATA[764,16] := 1.0;
   DATA[764,17] := 1.0;
   DATA[764,18] := 1.0;
   DATA[764,19] := 1.0;
   DATA[764,20] := 148.808;
   DATA[764,21] := 155.5242;
   DATA[764,22] := 1.718771;
   DATA[764,23] := 989.4001;
   DATA[764,24] := 2.0;
   DATA[764,25] := 2.0;
   DATA[764,26] := 7.878942;
   DATA[764,27] := 144.8603;
   DATA[764,28] := 263.1056;
   DATA[764,29] := 11.95847;
   DATA[764,30] := 1.730838;
   DATA[764,31] := 1.28167;
   DATA[764,32] := 0.7352687;
   DATA[764,33] := 0.3066329;
   DATA[764,34] := 2.0;
   DATA[764,35] := 250.8652;
   DATA[764,36] := 1.537821;
   DATA[764,37] := 189.6629;
   DATA[764,38] := 0.000128152;
   DATA[764,39] := 1.0;
   DATA[765,0] := 2.533068;
   DATA[765,1] := 544.0432;
   DATA[765,2] := 2.0;
   DATA[765,3] := 1.0;
   DATA[765,4] := 262.1764;
   DATA[765,5] := 8.412458;
   DATA[765,6] := 322.6096;
   DATA[765,7] := 0.000512607;
   DATA[765,8] := 1.0;
   DATA[765,9] := 1.0;
   DATA[765,10] := 1.0;
   DATA[765,11] := 2.013573;
   DATA[765,13] := 1009.076;
   DATA[765,14] := 1.0;
   DATA[765,15] := 1.0;
   DATA[765,16] := 1.0;
   DATA[765,17] := 1.0;
   DATA[765,18] := 1.0;
   DATA[765,19] := 1.0;
   DATA[765,20] := 148.808;
   DATA[765,21] := 155.5242;
   DATA[765,22] := 1.717233;
   DATA[765,23] := 989.3232;
   DATA[765,24] := 2.0;
   DATA[765,25] := 2.0;
   DATA[765,26] := 7.878942;
   DATA[765,27] := 144.8603;
   DATA[765,28] := 263.1056;
   DATA[765,29] := 11.95847;
   DATA[765,30] := 1.730069;
   DATA[765,31] := 1.28167;
   DATA[765,32] := 0.7352687;
   DATA[765,33] := 0.3066329;
   DATA[765,34] := 2.0;
   DATA[765,35] := 250.8652;
   DATA[765,36] := 1.665972;
   DATA[765,37] := 189.5828;
   DATA[765,38] := 0.000128152;
   DATA[765,39] := 1.0;
   DATA[766,0] := 2.533068;
   DATA[766,1] := 544.7498;
   DATA[766,2] := 2.0;
   DATA[766,3] := 1.0;
   DATA[766,4] := 262.1764;
   DATA[766,5] := 8.417906;
   DATA[766,6] := 321.8405;
   DATA[766,7] := 0.000512607;
   DATA[766,8] := 1.0;
   DATA[766,9] := 1.0;
   DATA[766,10] := 1.0;
   DATA[766,11] := 2.013573;
   DATA[766,13] := 1008.916;
   DATA[766,14] := 1.0;
   DATA[766,15] := 1.0;
   DATA[766,16] := 1.0;
   DATA[766,17] := 1.0;
   DATA[766,18] := 1.0;
   DATA[766,19] := 1.0;
   DATA[766,20] := 148.808;
   DATA[766,21] := 155.5242;
   DATA[766,22] := 1.717233;
   DATA[766,23] := 989.2848;
   DATA[766,24] := 2.0;
   DATA[766,25] := 2.0;
   DATA[766,26] := 7.878942;
   DATA[766,27] := 144.8603;
   DATA[766,28] := 263.1056;
   DATA[766,29] := 11.95847;
   DATA[766,30] := 1.728275;
   DATA[766,31] := 1.28167;
   DATA[766,32] := 0.7352687;
   DATA[766,33] := 0.3066329;
   DATA[766,34] := 2.0;
   DATA[766,35] := 250.8652;
   DATA[766,36] := 1.69801;
   DATA[766,37] := 189.5828;
   DATA[766,38] := 0.000128152;
   DATA[766,39] := 1.0;
   DATA[767,0] := 2.531467;
   DATA[767,1] := 545.4563;
   DATA[767,2] := 2.0;
   DATA[767,3] := 1.0;
   DATA[767,4] := 262.1764;
   DATA[767,5] := 8.422392;
   DATA[767,6] := 321.4048;
   DATA[767,8] := 1.0;
   DATA[767,9] := 1.0;
   DATA[767,10] := 1.0;
   DATA[767,11] := 2.013573;
   DATA[767,13] := 1009.637;
   DATA[767,14] := 1.0;
   DATA[767,15] := 1.0;
   DATA[767,16] := 1.0;
   DATA[767,17] := 1.0;
   DATA[767,18] := 1.0;
   DATA[767,19] := 1.0;
   DATA[767,20] := 148.808;
   DATA[767,21] := 155.5242;
   DATA[767,22] := 1.717233;
   DATA[767,23] := 988.5157;
   DATA[767,24] := 2.0;
   DATA[767,25] := 2.0;
   DATA[767,26] := 7.878942;
   DATA[767,27] := 144.8603;
   DATA[767,28] := 263.1056;
   DATA[767,29] := 11.95847;
   DATA[767,30] := 1.728275;
   DATA[767,31] := 1.294479;
   DATA[767,32] := 0.7352687;
   DATA[767,33] := 0.3066329;
   DATA[767,34] := 2.0;
   DATA[767,35] := 250.7049;
   DATA[767,36] := 1.69801;
   DATA[767,37] := 189.4066;
   DATA[767,38] := 0.000128152;
   DATA[767,39] := 1.0;
   DATA[768,0] := 2.531467;
   DATA[768,1] := 546.3199;
   DATA[768,2] := 2.0;
   DATA[768,3] := 1.0;
   DATA[768,4] := 262.1764;
   DATA[768,5] := 8.422712;
   DATA[768,6] := 320.8665;
   DATA[768,8] := 1.0;
   DATA[768,9] := 1.0;
   DATA[768,10] := 1.0;
   DATA[768,11] := 2.013573;
   DATA[768,13] := 1009.637;
   DATA[768,14] := 1.0;
   DATA[768,15] := 1.0;
   DATA[768,16] := 1.0;
   DATA[768,17] := 1.0;
   DATA[768,18] := 1.0;
   DATA[768,19] := 1.0;
   DATA[768,20] := 148.808;
   DATA[768,21] := 155.5242;
   DATA[768,22] := 1.717233;
   DATA[768,23] := 988.0543;
   DATA[768,24] := 2.0;
   DATA[768,25] := 2.0;
   DATA[768,26] := 7.878942;
   DATA[768,27] := 144.8603;
   DATA[768,28] := 263.1056;
   DATA[768,29] := 11.95847;
   DATA[768,30] := 1.728275;
   DATA[768,31] := 1.294479;
   DATA[768,32] := 0.7352687;
   DATA[768,33] := 0.3066329;
   DATA[768,34] := 2.0;
   DATA[768,35] := 250.6248;
   DATA[768,36] := 1.69801;
   DATA[768,37] := 189.3265;
   DATA[768,38] := 0.000128152;
   DATA[768,39] := 1.0;
   DATA[769,0] := 2.531467;
   DATA[769,1] := 546.4376;
   DATA[769,2] := 2.0;
   DATA[769,3] := 1.0;
   DATA[769,4] := 262.1764;
   DATA[769,5] := 8.425276;
   DATA[769,6] := 320.687;
   DATA[769,8] := 1.0;
   DATA[769,9] := 1.0;
   DATA[769,10] := 1.0;
   DATA[769,11] := 2.013573;
   DATA[769,13] := 1009.917;
   DATA[769,14] := 1.0;
   DATA[769,15] := 1.0;
   DATA[769,16] := 1.0;
   DATA[769,17] := 1.0;
   DATA[769,18] := 1.0;
   DATA[769,19] := 1.0;
   DATA[769,20] := 148.808;
   DATA[769,21] := 155.5242;
   DATA[769,22] := 1.717233;
   DATA[769,23] := 987.5544;
   DATA[769,24] := 2.0;
   DATA[769,25] := 2.0;
   DATA[769,26] := 7.878942;
   DATA[769,27] := 144.9116;
   DATA[769,28] := 263.1056;
   DATA[769,29] := 11.95847;
   DATA[769,30] := 1.728275;
   DATA[769,31] := 1.291533;
   DATA[769,32] := 0.7352687;
   DATA[769,33] := 0.3074016;
   DATA[769,34] := 2.0;
   DATA[769,35] := 250.6248;
   DATA[769,36] := 1.69801;
   DATA[769,37] := 189.3265;
   DATA[769,38] := 0.000128152;
   DATA[769,39] := 1.0;
   DATA[770,0] := 2.53435;
   DATA[770,1] := 546.6732;
   DATA[770,2] := 2.0;
   DATA[770,3] := 1.0;
   DATA[770,4] := 262.1764;
   DATA[770,5] := 8.432005;
   DATA[770,6] := 320.2512;
   DATA[770,8] := 1.0;
   DATA[770,9] := 1.0;
   DATA[770,10] := 1.0;
   DATA[770,11] := 2.013573;
   DATA[770,13] := 1009.877;
   DATA[770,14] := 1.0;
   DATA[770,15] := 1.0;
   DATA[770,16] := 1.0;
   DATA[770,17] := 1.0;
   DATA[770,18] := 1.0;
   DATA[770,19] := 1.0;
   DATA[770,20] := 148.808;
   DATA[770,21] := 155.5242;
   DATA[770,22] := 1.715952;
   DATA[770,23] := 987.1315;
   DATA[770,24] := 2.0;
   DATA[770,25] := 2.0;
   DATA[770,26] := 7.878942;
   DATA[770,27] := 144.9628;
   DATA[770,28] := 263.1056;
   DATA[770,29] := 11.95847;
   DATA[770,30] := 1.728275;
   DATA[770,31] := 1.290765;
   DATA[770,32] := 0.7352687;
   DATA[770,33] := 0.3074016;
   DATA[770,34] := 2.0;
   DATA[770,35] := 250.785;
   DATA[770,36] := 1.69801;
   DATA[770,37] := 189.5027;
   DATA[770,38] := 0.000128152;
   DATA[770,39] := 1.0;
   DATA[771,0] := 2.53435;
   DATA[771,1] := 546.6732;
   DATA[771,2] := 2.0;
   DATA[771,3] := 1.0;
   DATA[771,4] := 262.1764;
   DATA[771,5] := 8.432005;
   DATA[771,6] := 320.2512;
   DATA[771,8] := 1.0;
   DATA[771,9] := 1.0;
   DATA[771,10] := 1.0;
   DATA[771,11] := 2.013573;
   DATA[771,13] := 1009.877;
   DATA[771,14] := 1.0;
   DATA[771,15] := 1.0;
   DATA[771,16] := 1.0;
   DATA[771,17] := 1.0;
   DATA[771,18] := 1.0;
   DATA[771,19] := 1.0;
   DATA[771,20] := 148.808;
   DATA[771,21] := 155.5242;
   DATA[771,22] := 1.715952;
   DATA[771,23] := 987.1315;
   DATA[771,24] := 2.0;
   DATA[771,25] := 2.0;
   DATA[771,26] := 7.878942;
   DATA[771,27] := 144.9628;
   DATA[771,28] := 263.1056;
   DATA[771,29] := 11.95847;
   DATA[771,30] := 1.728275;
   DATA[771,31] := 1.290765;
   DATA[771,32] := 0.7352687;
   DATA[771,33] := 0.3074016;
   DATA[771,34] := 2.0;
   DATA[771,35] := 250.785;
   DATA[771,36] := 1.69801;
   DATA[771,37] := 189.5027;
   DATA[771,38] := 0.000128152;
   DATA[771,39] := 1.0;
   DATA[772,0] := 2.537232;
   DATA[772,1] := 546.5947;
   DATA[772,2] := 2.0;
   DATA[772,3] := 1.0;
   DATA[772,4] := 262.1764;
   DATA[772,5] := 8.432005;
   DATA[772,6] := 319.5847;
   DATA[772,8] := 1.0;
   DATA[772,9] := 1.0;
   DATA[772,10] := 1.0;
   DATA[772,11] := 2.013573;
   DATA[772,13] := 1010.038;
   DATA[772,14] := 1.0;
   DATA[772,15] := 1.0;
   DATA[772,16] := 1.0;
   DATA[772,17] := 1.0;
   DATA[772,18] := 1.0;
   DATA[772,19] := 1.0;
   DATA[772,20] := 148.808;
   DATA[772,21] := 155.5242;
   DATA[772,22] := 1.715952;
   DATA[772,23] := 986.747;
   DATA[772,24] := 2.0;
   DATA[772,25] := 2.0;
   DATA[772,26] := 7.878942;
   DATA[772,27] := 144.9628;
   DATA[772,28] := 263.1056;
   DATA[772,29] := 11.95847;
   DATA[772,30] := 1.728275;
   DATA[772,31] := 1.282183;
   DATA[772,32] := 0.7352687;
   DATA[772,33] := 0.3074016;
   DATA[772,34] := 2.0;
   DATA[772,35] := 250.9613;
   DATA[772,36] := 1.69801;
   DATA[772,37] := 189.6949;
   DATA[772,38] := 0.000128152;
   DATA[772,39] := 1.0;
   DATA[773,0] := 2.537232;
   DATA[773,1] := 546.6339;
   DATA[773,2] := 2.0;
   DATA[773,3] := 1.0;
   DATA[773,4] := 262.1764;
   DATA[773,5] := 8.434568;
   DATA[773,6] := 319.5847;
   DATA[773,8] := 1.0;
   DATA[773,9] := 1.0;
   DATA[773,10] := 1.0;
   DATA[773,11] := 2.013573;
   DATA[773,13] := 1009.917;
   DATA[773,14] := 1.0;
   DATA[773,15] := 1.0;
   DATA[773,16] := 1.0;
   DATA[773,17] := 1.0;
   DATA[773,18] := 1.0;
   DATA[773,19] := 1.0;
   DATA[773,20] := 148.808;
   DATA[773,21] := 155.5242;
   DATA[773,22] := 1.715952;
   DATA[773,23] := 986.2087;
   DATA[773,24] := 2.0;
   DATA[773,25] := 2.0;
   DATA[773,26] := 7.878942;
   DATA[773,27] := 144.9628;
   DATA[773,28] := 263.1056;
   DATA[773,29] := 11.95847;
   DATA[773,30] := 1.728788;
   DATA[773,31] := 1.290252;
   DATA[773,32] := 0.7352687;
   DATA[773,33] := 0.3065048;
   DATA[773,34] := 2.0;
   DATA[773,35] := 250.9613;
   DATA[773,36] := 1.649953;
   DATA[773,37] := 189.759;
   DATA[773,38] := 0.000128152;
   DATA[773,39] := 1.0;
   DATA[774,0] := 2.537232;
   DATA[774,1] := 547.0264;
   DATA[774,2] := 2.0;
   DATA[774,3] := 1.0;
   DATA[774,4] := 262.1764;
   DATA[774,5] := 8.439695;
   DATA[774,6] := 318.9695;
   DATA[774,8] := 1.0;
   DATA[774,9] := 1.0;
   DATA[774,10] := 1.0;
   DATA[774,11] := 2.013573;
   DATA[774,13] := 1009.757;
   DATA[774,14] := 1.0;
   DATA[774,15] := 1.0;
   DATA[774,16] := 1.0;
   DATA[774,17] := 1.0;
   DATA[774,18] := 1.0;
   DATA[774,19] := 1.0;
   DATA[774,20] := 148.808;
   DATA[774,21] := 155.6524;
   DATA[774,22] := 1.717746;
   DATA[774,23] := 986.0164;
   DATA[774,24] := 2.0;
   DATA[774,25] := 2.0;
   DATA[774,26] := 7.878942;
   DATA[774,27] := 144.9628;
   DATA[774,28] := 263.1056;
   DATA[774,29] := 11.95847;
   DATA[774,30] := 1.731864;
   DATA[774,31] := 1.297554;
   DATA[774,32] := 0.7352687;
   DATA[774,33] := 0.3065048;
   DATA[774,34] := 2.0;
   DATA[774,35] := 250.9613;
   DATA[774,36] := 1.649953;
   DATA[774,37] := 189.759;
   DATA[774,38] := 0.000128152;
   DATA[774,39] := 1.0;
   DATA[775,0] := 2.537232;
   DATA[775,1] := 546.9872;
   DATA[775,2] := 2.0;
   DATA[775,3] := 1.0;
   DATA[775,4] := 262.1764;
   DATA[775,5] := 8.4429;
   DATA[775,6] := 318.9695;
   DATA[775,8] := 1.0;
   DATA[775,9] := 1.0;
   DATA[775,10] := 1.0;
   DATA[775,11] := 2.013573;
   DATA[775,13] := 1010.078;
   DATA[775,14] := 1.0;
   DATA[775,15] := 1.0;
   DATA[775,16] := 1.0;
   DATA[775,17] := 1.0;
   DATA[775,18] := 1.0;
   DATA[775,19] := 1.0;
   DATA[775,20] := 148.808;
   DATA[775,21] := 155.6524;
   DATA[775,22] := 1.717746;
   DATA[775,23] := 985.5934;
   DATA[775,24] := 2.0;
   DATA[775,25] := 2.0;
   DATA[775,26] := 7.878942;
   DATA[775,27] := 144.9628;
   DATA[775,28] := 263.1056;
   DATA[775,29] := 11.95847;
   DATA[775,30] := 1.731864;
   DATA[775,31] := 1.308569;
   DATA[775,32] := 0.7352687;
   DATA[775,33] := 0.3065048;
   DATA[775,34] := 2.0;
   DATA[775,35] := 250.9613;
   DATA[775,36] := 1.649953;
   DATA[775,37] := 189.759;
   DATA[775,38] := 0.000128152;
   DATA[775,39] := 1.0;
   DATA[776,0] := 2.537232;
   DATA[776,1] := 546.8694;
   DATA[776,2] := 2.0;
   DATA[776,3] := 1.0;
   DATA[776,4] := 262.1764;
   DATA[776,5] := 8.4429;
   DATA[776,6] := 318.8926;
   DATA[776,8] := 1.0;
   DATA[776,9] := 1.0;
   DATA[776,10] := 1.0;
   DATA[776,11] := 2.013573;
   DATA[776,13] := 1010.638;
   DATA[776,14] := 1.0;
   DATA[776,15] := 1.0;
   DATA[776,16] := 1.0;
   DATA[776,17] := 1.0;
   DATA[776,18] := 1.0;
   DATA[776,19] := 1.0;
   DATA[776,20] := 148.808;
   DATA[776,21] := 155.7293;
   DATA[776,22] := 1.717746;
   DATA[776,23] := 985.2089;
   DATA[776,24] := 2.0;
   DATA[776,25] := 2.0;
   DATA[776,26] := 7.878942;
   DATA[776,27] := 144.9628;
   DATA[776,28] := 263.1056;
   DATA[776,29] := 11.95847;
   DATA[776,30] := 1.731864;
   DATA[776,31] := 1.318432;
   DATA[776,32] := 0.7352687;
   DATA[776,33] := 0.3065048;
   DATA[776,34] := 2.0;
   DATA[776,35] := 250.9613;
   DATA[776,36] := 1.649953;
   DATA[776,37] := 189.759;
   DATA[776,38] := 0.000128152;
   DATA[776,39] := 1.0;
   DATA[777,0] := 2.542677;
   DATA[777,1] := 547.262;
   DATA[777,2] := 2.0;
   DATA[777,3] := 1.0;
   DATA[777,4] := 262.1764;
   DATA[777,5] := 8.444822;
   DATA[777,6] := 318.3799;
   DATA[777,8] := 1.0;
   DATA[777,9] := 1.0;
   DATA[777,10] := 1.0;
   DATA[777,11] := 2.013573;
   DATA[777,13] := 1010.839;
   DATA[777,14] := 1.0;
   DATA[777,15] := 1.0;
   DATA[777,16] := 1.0;
   DATA[777,17] := 1.0;
   DATA[777,18] := 1.0;
   DATA[777,19] := 1.0;
   DATA[777,20] := 148.808;
   DATA[777,21] := 155.7293;
   DATA[777,22] := 1.717361;
   DATA[777,23] := 984.5937;
   DATA[777,24] := 2.0;
   DATA[777,25] := 2.0;
   DATA[777,26] := 7.878942;
   DATA[777,27] := 144.9628;
   DATA[777,28] := 263.1056;
   DATA[777,29] := 11.95847;
   DATA[777,30] := 1.731864;
   DATA[777,31] := 1.321506;
   DATA[777,32] := 0.7352687;
   DATA[777,33] := 0.3065048;
   DATA[777,34] := 2.0;
   DATA[777,35] := 251.1055;
   DATA[777,36] := 1.649953;
   DATA[777,37] := 189.759;
   DATA[777,38] := 0.000128152;
   DATA[777,39] := 1.0;
   DATA[778,0] := 2.543958;
   DATA[778,1] := 547.6152;
   DATA[778,2] := 2.0;
   DATA[778,3] := 1.0;
   DATA[778,4] := 262.1764;
   DATA[778,5] := 8.449949;
   DATA[778,6] := 318.2774;
   DATA[778,8] := 1.0;
   DATA[778,9] := 1.0;
   DATA[778,10] := 1.0;
   DATA[778,11] := 2.013573;
   DATA[778,13] := 1010.758;
   DATA[778,14] := 1.0;
   DATA[778,15] := 1.0;
   DATA[778,16] := 1.0;
   DATA[778,17] := 1.0;
   DATA[778,18] := 1.0;
   DATA[778,19] := 1.0;
   DATA[778,20] := 148.808;
   DATA[778,21] := 155.7293;
   DATA[778,22] := 1.717233;
   DATA[778,23] := 984.4014;
   DATA[778,24] := 2.0;
   DATA[778,25] := 2.0;
   DATA[778,26] := 7.878942;
   DATA[778,27] := 144.9628;
   DATA[778,28] := 263.1056;
   DATA[778,29] := 11.95847;
   DATA[778,30] := 1.731864;
   DATA[778,31] := 1.31254;
   DATA[778,32] := 0.7352687;
   DATA[778,33] := 0.3065048;
   DATA[778,34] := 2.0;
   DATA[778,35] := 251.1055;
   DATA[778,36] := 1.649953;
   DATA[778,37] := 189.759;
   DATA[778,38] := 0.000128152;
   DATA[778,39] := 1.0;
   DATA[779,0] := 2.543958;
   DATA[779,1] := 547.4975;
   DATA[779,2] := 2.0;
   DATA[779,3] := 1.0;
   DATA[779,4] := 262.1764;
   DATA[779,5] := 8.452192;
   DATA[779,6] := 317.9954;
   DATA[779,8] := 1.0;
   DATA[779,9] := 1.0;
   DATA[779,10] := 1.0;
   DATA[779,11] := 2.013573;
   DATA[779,13] := 1010.758;
   DATA[779,14] := 1.0;
   DATA[779,15] := 1.0;
   DATA[779,16] := 1.0;
   DATA[779,17] := 1.0;
   DATA[779,18] := 1.0;
   DATA[779,19] := 1.0;
   DATA[779,20] := 148.808;
   DATA[779,21] := 155.7293;
   DATA[779,22] := 1.717233;
   DATA[779,23] := 983.7862;
   DATA[779,24] := 2.0;
   DATA[779,25] := 2.0;
   DATA[779,26] := 7.878942;
   DATA[779,27] := 144.9628;
   DATA[779,28] := 263.1056;
   DATA[779,29] := 11.95847;
   DATA[779,30] := 1.731864;
   DATA[779,31] := 1.304214;
   DATA[779,32] := 0.7352687;
   DATA[779,33] := 0.3065048;
   DATA[779,34] := 2.0;
   DATA[779,35] := 251.1055;
   DATA[779,36] := 1.649953;
   DATA[779,37] := 189.759;
   DATA[779,38] := 0.000128152;
   DATA[779,39] := 1.0;
   DATA[780,0] := 2.543958;
   DATA[780,1] := 547.4582;
   DATA[780,2] := 2.0;
   DATA[780,3] := 1.0;
   DATA[780,4] := 262.1764;
   DATA[780,5] := 8.452833;
   DATA[780,6] := 317.9185;
   DATA[780,8] := 1.0;
   DATA[780,9] := 1.0;
   DATA[780,10] := 1.0;
   DATA[780,11] := 2.013573;
   DATA[780,13] := 1010.638;
   DATA[780,14] := 1.0;
   DATA[780,15] := 1.0;
   DATA[780,16] := 1.0;
   DATA[780,17] := 1.0;
   DATA[780,18] := 1.0;
   DATA[780,19] := 1.0;
   DATA[780,20] := 148.808;
   DATA[780,21] := 155.7293;
   DATA[780,22] := 1.717233;
   DATA[780,23] := 983.5939;
   DATA[780,24] := 2.0;
   DATA[780,25] := 2.0;
   DATA[780,26] := 7.878942;
   DATA[780,27] := 144.9628;
   DATA[780,28] := 263.1056;
   DATA[780,29] := 11.95847;
   DATA[780,30] := 1.730582;
   DATA[780,31] := 1.297682;
   DATA[780,32] := 0.7352687;
   DATA[780,33] := 0.3065048;
   DATA[780,34] := 2.0;
   DATA[780,35] := 251.1055;
   DATA[780,36] := 1.649953;
   DATA[780,37] := 189.759;
   DATA[780,38] := 0.000128152;
   DATA[780,39] := 1.0;
   DATA[781,0] := 2.539474;
   DATA[781,1] := 547.4189;
   DATA[781,2] := 2.0;
   DATA[781,3] := 1.0;
   DATA[781,4] := 262.1764;
   DATA[781,5] := 8.452833;
   DATA[781,6] := 317.8672;
   DATA[781,8] := 1.0;
   DATA[781,9] := 1.0;
   DATA[781,10] := 1.0;
   DATA[781,11] := 2.013573;
   DATA[781,13] := 1010.758;
   DATA[781,14] := 1.0;
   DATA[781,15] := 1.0;
   DATA[781,16] := 1.0;
   DATA[781,17] := 1.0;
   DATA[781,18] := 1.0;
   DATA[781,19] := 1.0;
   DATA[781,20] := 148.808;
   DATA[781,21] := 155.7293;
   DATA[781,22] := 1.717233;
   DATA[781,23] := 983.0556;
   DATA[781,24] := 2.0;
   DATA[781,25] := 2.0;
   DATA[781,26] := 7.878942;
   DATA[781,27] := 144.9628;
   DATA[781,28] := 263.1056;
   DATA[781,29] := 11.95847;
   DATA[781,30] := 1.730582;
   DATA[781,31] := 1.291533;
   DATA[781,32] := 0.7352687;
   DATA[781,33] := 0.3065048;
   DATA[781,34] := 2.0;
   DATA[781,35] := 251.1055;
   DATA[781,36] := 1.69801;
   DATA[781,37] := 189.759;
   DATA[781,38] := 0.000128152;
   DATA[781,39] := 1.0;
   DATA[782,0] := 2.537873;
   DATA[782,1] := 547.9685;
   DATA[782,2] := 2.0;
   DATA[782,3] := 1.0;
   DATA[782,4] := 262.1764;
   DATA[782,5] := 8.456038;
   DATA[782,6] := 317.7903;
   DATA[782,8] := 1.0;
   DATA[782,9] := 1.0;
   DATA[782,10] := 1.0;
   DATA[782,11] := 2.042384;
   DATA[782,13] := 1010.438;
   DATA[782,14] := 1.0;
   DATA[782,15] := 1.0;
   DATA[782,16] := 1.0;
   DATA[782,17] := 1.0;
   DATA[782,18] := 1.0;
   DATA[782,19] := 1.0;
   DATA[782,20] := 148.808;
   DATA[782,21] := 155.7293;
   DATA[782,22] := 1.717233;
   DATA[782,23] := 982.4789;
   DATA[782,24] := 2.0;
   DATA[782,25] := 2.0;
   DATA[782,26] := 7.878942;
   DATA[782,27] := 144.9628;
   DATA[782,28] := 263.1056;
   DATA[782,29] := 11.95847;
   DATA[782,30] := 1.730582;
   DATA[782,31] := 1.291533;
   DATA[782,32] := 0.7352687;
   DATA[782,33] := 0.3065048;
   DATA[782,34] := 2.0;
   DATA[782,35] := 251.1055;
   DATA[782,36] := 1.69801;
   DATA[782,37] := 189.759;
   DATA[782,38] := 0.000128152;
   DATA[782,39] := 1.0;
   DATA[783,0] := 2.537873;
   DATA[783,1] := 548.9891;
   DATA[783,2] := 2.0;
   DATA[783,3] := 1.0;
   DATA[783,4] := 262.1764;
   DATA[783,5] := 8.456038;
   DATA[783,6] := 317.6109;
   DATA[783,8] := 1.0;
   DATA[783,9] := 1.0;
   DATA[783,10] := 1.0;
   DATA[783,11] := 2.042384;
   DATA[783,13] := 1010.518;
   DATA[783,14] := 1.0;
   DATA[783,15] := 1.0;
   DATA[783,16] := 1.0;
   DATA[783,17] := 1.0;
   DATA[783,18] := 1.0;
   DATA[783,19] := 1.0;
   DATA[783,20] := 148.808;
   DATA[783,21] := 155.7293;
   DATA[783,22] := 1.720309;
   DATA[783,23] := 982.4404;
   DATA[783,24] := 2.0;
   DATA[783,25] := 2.0;
   DATA[783,26] := 7.878942;
   DATA[783,27] := 144.9628;
   DATA[783,28] := 263.1056;
   DATA[783,29] := 11.95847;
   DATA[783,30] := 1.728788;
   DATA[783,31] := 1.295888;
   DATA[783,32] := 0.7352687;
   DATA[783,33] := 0.3065048;
   DATA[783,34] := 2.0;
   DATA[783,35] := 251.1055;
   DATA[783,36] := 1.69801;
   DATA[783,37] := 189.759;
   DATA[783,38] := 0.000128152;
   DATA[783,39] := 1.0;
   DATA[784,0] := 2.533709;
   DATA[784,1] := 549.7349;
   DATA[784,2] := 2.0;
   DATA[784,3] := 1.0;
   DATA[784,4] := 262.1764;
   DATA[784,5] := 8.456038;
   DATA[784,6] := 317.5083;
   DATA[784,8] := 1.0;
   DATA[784,9] := 1.0;
   DATA[784,10] := 1.0;
   DATA[784,11] := 2.042384;
   DATA[784,13] := 1010.678;
   DATA[784,14] := 1.0;
   DATA[784,15] := 1.0;
   DATA[784,16] := 1.0;
   DATA[784,17] := 1.0;
   DATA[784,18] := 1.0;
   DATA[784,19] := 1.0;
   DATA[784,20] := 148.808;
   DATA[784,21] := 155.7293;
   DATA[784,22] := 1.720309;
   DATA[784,23] := 982.2482;
   DATA[784,24] := 2.0;
   DATA[784,25] := 2.0;
   DATA[784,26] := 7.878942;
   DATA[784,27] := 144.9628;
   DATA[784,28] := 263.1056;
   DATA[784,29] := 11.95847;
   DATA[784,30] := 1.728788;
   DATA[784,31] := 1.291405;
   DATA[784,32] := 0.7352687;
   DATA[784,33] := 0.3065048;
   DATA[784,34] := 2.0;
   DATA[784,35] := 250.9613;
   DATA[784,36] := 1.69801;
   DATA[784,37] := 189.759;
   DATA[784,38] := 0.000128152;
   DATA[784,39] := 1.0;
   DATA[785,0] := 2.533709;
   DATA[785,1] := 549.6564;
   DATA[785,2] := 2.0;
   DATA[785,3] := 1.0;
   DATA[785,4] := 262.1764;
   DATA[785,5] := 8.45764;
   DATA[785,6] := 317.252;
   DATA[785,8] := 1.0;
   DATA[785,9] := 1.0;
   DATA[785,10] := 1.0;
   DATA[785,11] := 2.042384;
   DATA[785,13] := 1010.839;
   DATA[785,14] := 1.0;
   DATA[785,15] := 1.0;
   DATA[785,16] := 1.0;
   DATA[785,17] := 1.0;
   DATA[785,18] := 1.0;
   DATA[785,19] := 1.0;
   DATA[785,20] := 148.808;
   DATA[785,21] := 155.7293;
   DATA[785,22] := 1.720309;
   DATA[785,23] := 981.979;
   DATA[785,24] := 2.0;
   DATA[785,25] := 2.0;
   DATA[785,26] := 7.878942;
   DATA[785,27] := 144.9628;
   DATA[785,28] := 263.1056;
   DATA[785,29] := 11.95847;
   DATA[785,30] := 1.728788;
   DATA[785,31] := 1.282311;
   DATA[785,32] := 0.7352687;
   DATA[785,33] := 0.3065048;
   DATA[785,34] := 2.0;
   DATA[785,35] := 250.9453;
   DATA[785,36] := 1.69801;
   DATA[785,37] := 189.759;
   DATA[785,38] := 0.000128152;
   DATA[785,39] := 1.0;
   DATA[786,0] := 2.537232;
   DATA[786,1] := 550.4414;
   DATA[786,2] := 2.0;
   DATA[786,3] := 1.0;
   DATA[786,4] := 262.1764;
   DATA[786,5] := 8.461805;
   DATA[786,6] := 317.1751;
   DATA[786,8] := 1.0;
   DATA[786,9] := 1.0;
   DATA[786,10] := 1.0;
   DATA[786,11] := 2.042384;
   DATA[786,13] := 1010.678;
   DATA[786,14] := 1.0;
   DATA[786,15] := 1.0;
   DATA[786,16] := 1.0;
   DATA[786,17] := 1.0;
   DATA[786,18] := 1.0;
   DATA[786,19] := 1.0;
   DATA[786,20] := 148.808;
   DATA[786,21] := 155.5242;
   DATA[786,22] := 1.718002;
   DATA[786,23] := 981.7483;
   DATA[786,24] := 2.0;
   DATA[786,25] := 2.0;
   DATA[786,26] := 7.878942;
   DATA[786,27] := 144.9628;
   DATA[786,28] := 263.1056;
   DATA[786,29] := 11.95847;
   DATA[786,30] := 1.729428;
   DATA[786,31] := 1.286666;
   DATA[786,32] := 0.7352687;
   DATA[786,33] := 0.3065048;
   DATA[786,34] := 2.0;
   DATA[786,35] := 250.9453;
   DATA[786,36] := 1.746067;
   DATA[786,37] := 189.743;
   DATA[786,38] := 0.000128152;
   DATA[786,39] := 1.0;
   DATA[787,0] := 2.540115;
   DATA[787,1] := 551.1087;
   DATA[787,2] := 2.0;
   DATA[787,3] := 1.0;
   DATA[787,4] := 262.1764;
   DATA[787,5] := 8.461805;
   DATA[787,6] := 317.1751;
   DATA[787,8] := 1.0;
   DATA[787,9] := 1.0;
   DATA[787,10] := 1.0;
   DATA[787,11] := 2.042384;
   DATA[787,13] := 1010.638;
   DATA[787,14] := 1.0;
   DATA[787,15] := 1.0;
   DATA[787,16] := 1.0;
   DATA[787,17] := 1.0;
   DATA[787,18] := 1.0;
   DATA[787,19] := 1.0;
   DATA[787,20] := 148.808;
   DATA[787,21] := 155.5242;
   DATA[787,22] := 1.717874;
   DATA[787,23] := 981.3638;
   DATA[787,24] := 2.0;
   DATA[787,25] := 2.0;
   DATA[787,26] := 7.878942;
   DATA[787,27] := 144.9628;
   DATA[787,28] := 263.1056;
   DATA[787,29] := 11.95847;
   DATA[787,30] := 1.730197;
   DATA[787,31] := 1.280646;
   DATA[787,32] := 0.7352687;
   DATA[787,33] := 0.3065048;
   DATA[787,34] := 2.0;
   DATA[787,35] := 250.9453;
   DATA[787,36] := 1.746067;
   DATA[787,37] := 189.743;
   DATA[787,38] := 0.000128152;
   DATA[787,39] := 1.0;
   DATA[788,0] := 2.54652;
   DATA[788,1] := 551.619;
   DATA[788,2] := 2.0;
   DATA[788,3] := 1.0;
   DATA[788,4] := 262.1764;
   DATA[788,5] := 8.461805;
   DATA[788,6] := 317.1751;
   DATA[788,8] := 1.0;
   DATA[788,9] := 1.0;
   DATA[788,10] := 1.0;
   DATA[788,11] := 2.042384;
   DATA[788,13] := 1010.718;
   DATA[788,14] := 1.0;
   DATA[788,15] := 1.0;
   DATA[788,16] := 1.0;
   DATA[788,17] := 1.0;
   DATA[788,18] := 1.0;
   DATA[788,19] := 1.0;
   DATA[788,20] := 148.808;
   DATA[788,21] := 155.5242;
   DATA[788,22] := 1.717874;
   DATA[788,23] := 981.0946;
   DATA[788,24] := 2.0;
   DATA[788,25] := 2.0;
   DATA[788,26] := 7.878942;
   DATA[788,27] := 144.9628;
   DATA[788,28] := 263.1056;
   DATA[788,29] := 11.95847;
   DATA[788,30] := 1.730197;
   DATA[788,31] := 1.291533;
   DATA[788,32] := 0.7352687;
   DATA[788,33] := 0.3065048;
   DATA[788,34] := 2.0;
   DATA[788,35] := 250.9453;
   DATA[788,36] := 1.746067;
   DATA[788,37] := 189.743;
   DATA[788,38] := 0.000128152;
   DATA[788,39] := 1.0;
   DATA[789,0] := 2.547161;
   DATA[789,1] := 552.3648;
   DATA[789,2] := 2.0;
   DATA[789,3] := 1.0;
   DATA[789,4] := 262.1764;
   DATA[789,5] := 8.461805;
   DATA[789,6] := 317.1751;
   DATA[789,8] := 1.0;
   DATA[789,9] := 1.0;
   DATA[789,10] := 1.0;
   DATA[789,11] := 2.042384;
   DATA[789,13] := 1010.558;
   DATA[789,14] := 1.0;
   DATA[789,15] := 1.0;
   DATA[789,16] := 1.0;
   DATA[789,17] := 1.0;
   DATA[789,18] := 1.0;
   DATA[789,19] := 1.0;
   DATA[789,20] := 148.808;
   DATA[789,21] := 155.678;
   DATA[789,22] := 1.717874;
   DATA[789,23] := 980.9408;
   DATA[789,24] := 2.0;
   DATA[789,25] := 2.0;
   DATA[789,26] := 7.878942;
   DATA[789,27] := 145.1166;
   DATA[789,28] := 263.1056;
   DATA[789,29] := 11.95847;
   DATA[789,30] := 1.730197;
   DATA[789,31] := 1.291789;
   DATA[789,32] := 0.7352687;
   DATA[789,33] := 0.306761;
   DATA[789,34] := 2.0;
   DATA[789,35] := 250.9453;
   DATA[789,36] := 1.746067;
   DATA[789,37] := 189.6469;
   DATA[789,38] := 0.000128152;
   DATA[789,39] := 1.0;
   DATA[790,0] := 2.548762;
   DATA[790,1] := 553.1106;
   DATA[790,2] := 2.0;
   DATA[790,3] := 1.0;
   DATA[790,4] := 262.1764;
   DATA[790,5] := 8.461805;
   DATA[790,6] := 316.8675;
   DATA[790,8] := 1.0;
   DATA[790,9] := 1.0;
   DATA[790,10] := 1.0;
   DATA[790,11] := 2.042384;
   DATA[790,13] := 1011.039;
   DATA[790,14] := 1.0;
   DATA[790,15] := 1.0;
   DATA[790,16] := 1.0;
   DATA[790,17] := 1.0;
   DATA[790,18] := 1.0;
   DATA[790,19] := 1.0;
   DATA[790,20] := 148.808;
   DATA[790,21] := 155.7293;
   DATA[790,22] := 1.717874;
   DATA[790,23] := 980.364;
   DATA[790,24] := 2.0;
   DATA[790,25] := 2.0;
   DATA[790,26] := 7.878942;
   DATA[790,27] := 145.1423;
   DATA[790,28] := 263.1056;
   DATA[790,29] := 11.95847;
   DATA[790,30] := 1.728531;
   DATA[790,31] := 1.281798;
   DATA[790,32] := 0.7352687;
   DATA[790,33] := 0.3069532;
   DATA[790,34] := 2.0;
   DATA[790,35] := 250.9453;
   DATA[790,36] := 1.746067;
   DATA[790,37] := 189.6469;
   DATA[790,38] := 0.000128152;
   DATA[790,39] := 1.0;
   DATA[791,0] := 2.550043;
   DATA[791,1] := 554.0527;
   DATA[791,2] := 2.0;
   DATA[791,3] := 1.0;
   DATA[791,4] := 262.1764;
   DATA[791,5] := 8.461805;
   DATA[791,6] := 316.8675;
   DATA[791,8] := 1.0;
   DATA[791,9] := 1.0;
   DATA[791,10] := 1.0;
   DATA[791,11] := 2.042384;
   DATA[791,13] := 1011.119;
   DATA[791,14] := 1.0;
   DATA[791,15] := 1.0;
   DATA[791,16] := 1.0;
   DATA[791,17] := 1.0;
   DATA[791,18] := 1.0;
   DATA[791,19] := 1.0;
   DATA[791,20] := 148.808;
   DATA[791,21] := 155.7293;
   DATA[791,22] := 1.717874;
   DATA[791,23] := 979.6719;
   DATA[791,24] := 2.0;
   DATA[791,25] := 2.0;
   DATA[791,26] := 7.878942;
   DATA[791,27] := 145.1423;
   DATA[791,28] := 263.1056;
   DATA[791,29] := 11.95847;
   DATA[791,30] := 1.728531;
   DATA[791,31] := 1.274625;
   DATA[791,32] := 0.7352687;
   DATA[791,33] := 0.3069532;
   DATA[791,34] := 2.0;
   DATA[791,35] := 250.9453;
   DATA[791,36] := 1.746067;
   DATA[791,37] := 189.6469;
   DATA[791,38] := 0.000128152;
   DATA[791,39] := 1.0;
   DATA[792,0] := 2.551965;
   DATA[792,1] := 554.6807;
   DATA[792,2] := 2.0;
   DATA[792,3] := 1.0;
   DATA[792,4] := 262.1764;
   DATA[792,5] := 8.46533;
   DATA[792,6] := 316.8675;
   DATA[792,8] := 1.0;
   DATA[792,9] := 1.0;
   DATA[792,10] := 1.0;
   DATA[792,11] := 2.042384;
   DATA[792,13] := 1011.159;
   DATA[792,14] := 1.0;
   DATA[792,15] := 1.0;
   DATA[792,16] := 1.0;
   DATA[792,17] := 1.0;
   DATA[792,18] := 1.0;
   DATA[792,19] := 1.0;
   DATA[792,20] := 148.808;
   DATA[792,21] := 155.7293;
   DATA[792,22] := 1.717874;
   DATA[792,23] := 979.4796;
   DATA[792,24] := 2.0;
   DATA[792,25] := 2.0;
   DATA[792,26] := 7.878942;
   DATA[792,27] := 145.1423;
   DATA[792,28] := 263.0415;
   DATA[792,29] := 11.95847;
   DATA[792,30] := 1.728531;
   DATA[792,31] := 1.263866;
   DATA[792,32] := 0.7352687;
   DATA[792,33] := 0.3069532;
   DATA[792,34] := 2.0;
   DATA[792,35] := 250.9453;
   DATA[792,36] := 1.746067;
   DATA[792,37] := 189.6469;
   DATA[792,38] := 0.000128152;
   DATA[792,39] := 1.0;
   DATA[793,0] := 2.552926;
   DATA[793,1] := 555.4265;
   DATA[793,2] := 2.0;
   DATA[793,3] := 1.0;
   DATA[793,4] := 262.1764;
   DATA[793,5] := 8.46533;
   DATA[793,6] := 316.7137;
   DATA[793,8] := 1.0;
   DATA[793,9] := 1.0;
   DATA[793,10] := 1.0;
   DATA[793,11] := 2.042384;
   DATA[793,13] := 1010.839;
   DATA[793,14] := 1.0;
   DATA[793,15] := 1.0;
   DATA[793,16] := 1.0;
   DATA[793,17] := 1.0;
   DATA[793,18] := 1.0;
   DATA[793,19] := 1.0;
   DATA[793,20] := 148.808;
   DATA[793,21] := 155.7293;
   DATA[793,22] := 1.717874;
   DATA[793,23] := 978.9797;
   DATA[793,24] := 2.0;
   DATA[793,25] := 2.0;
   DATA[793,26] := 7.878942;
   DATA[793,27] := 145.1423;
   DATA[793,28] := 263.0415;
   DATA[793,29] := 11.95847;
   DATA[793,30] := 1.728531;
   DATA[793,31] := 1.262713;
   DATA[793,32] := 0.7352687;
   DATA[793,33] := 0.3075937;
   DATA[793,34] := 2.0;
   DATA[793,35] := 250.8171;
   DATA[793,36] := 1.746067;
   DATA[793,37] := 189.6469;
   DATA[793,38] := 0.000128152;
   DATA[793,39] := 1.0;
   DATA[794,0] := 2.552926;
   DATA[794,1] := 555.819;
   DATA[794,2] := 2.0;
   DATA[794,3] := 1.0;
   DATA[794,4] := 262.1764;
   DATA[794,5] := 8.46533;
   DATA[794,6] := 316.5086;
   DATA[794,8] := 1.0;
   DATA[794,9] := 1.0;
   DATA[794,10] := 1.0;
   DATA[794,11] := 2.042384;
   DATA[794,13] := 1011.079;
   DATA[794,14] := 1.0;
   DATA[794,15] := 1.0;
   DATA[794,16] := 1.0;
   DATA[794,17] := 1.0;
   DATA[794,18] := 1.0;
   DATA[794,19] := 1.0;
   DATA[794,20] := 148.808;
   DATA[794,21] := 155.7293;
   DATA[794,22] := 1.717874;
   DATA[794,23] := 978.9797;
   DATA[794,24] := 2.0;
   DATA[794,25] := 2.0;
   DATA[794,26] := 7.878942;
   DATA[794,27] := 145.1166;
   DATA[794,28] := 263.0415;
   DATA[794,29] := 11.95847;
   DATA[794,30] := 1.726352;
   DATA[794,31] := 1.278084;
   DATA[794,32] := 0.7352687;
   DATA[794,33] := 0.3077859;
   DATA[794,34] := 2.0;
   DATA[794,35] := 250.8171;
   DATA[794,36] := 1.746067;
   DATA[794,37] := 189.6469;
   DATA[794,38] := 0.000128152;
   DATA[794,39] := 1.0;
   DATA[795,0] := 2.552926;
   DATA[795,1] := 556.1723;
   DATA[795,2] := 2.0;
   DATA[795,3] := 1.0;
   DATA[795,4] := 262.1764;
   DATA[795,5] := 8.46533;
   DATA[795,6] := 316.5086;
   DATA[795,8] := 1.0;
   DATA[795,9] := 1.0;
   DATA[795,10] := 1.0;
   DATA[795,11] := 2.042384;
   DATA[795,13] := 1010.518;
   DATA[795,14] := 1.0;
   DATA[795,15] := 1.0;
   DATA[795,16] := 1.0;
   DATA[795,17] := 1.0;
   DATA[795,18] := 1.0;
   DATA[795,19] := 1.0;
   DATA[795,20] := 148.808;
   DATA[795,21] := 155.7293;
   DATA[795,22] := 1.717874;
   DATA[795,23] := 978.8259;
   DATA[795,24] := 2.0;
   DATA[795,25] := 2.0;
   DATA[795,26] := 7.878942;
   DATA[795,27] := 144.9116;
   DATA[795,28] := 263.0415;
   DATA[795,29] := 11.95847;
   DATA[795,30] := 1.726352;
   DATA[795,31] := 1.289356;
   DATA[795,32] := 0.7352687;
   DATA[795,33] := 0.306761;
   DATA[795,34] := 2.0;
   DATA[795,35] := 250.8171;
   DATA[795,36] := 1.69801;
   DATA[795,37] := 189.6469;
   DATA[795,38] := 0.000128152;
   DATA[795,39] := 1.0;
   DATA[796,0] := 2.548442;
   DATA[796,1] := 556.5649;
   DATA[796,2] := 2.0;
   DATA[796,3] := 1.0;
   DATA[796,4] := 262.1764;
   DATA[796,5] := 8.46533;
   DATA[796,6] := 316.4573;
   DATA[796,8] := 1.0;
   DATA[796,9] := 1.0;
   DATA[796,10] := 1.0;
   DATA[796,11] := 2.042384;
   DATA[796,13] := 1010.959;
   DATA[796,14] := 1.0;
   DATA[796,15] := 1.0;
   DATA[796,16] := 1.0;
   DATA[796,17] := 1.0;
   DATA[796,18] := 1.0;
   DATA[796,19] := 1.0;
   DATA[796,20] := 148.808;
   DATA[796,21] := 155.7293;
   DATA[796,22] := 1.717874;
   DATA[796,23] := 978.9028;
   DATA[796,24] := 2.0;
   DATA[796,25] := 2.0;
   DATA[796,26] := 7.878942;
   DATA[796,27] := 144.9116;
   DATA[796,28] := 263.0415;
   DATA[796,29] := 11.95847;
   DATA[796,30] := 1.726352;
   DATA[796,31] := 1.300115;
   DATA[796,32] := 0.7352687;
   DATA[796,33] := 0.3066329;
   DATA[796,34] := 2.0;
   DATA[796,35] := 250.8171;
   DATA[796,36] := 1.69801;
   DATA[796,37] := 189.6469;
   DATA[796,38] := 0.000128152;
   DATA[796,39] := 1.0;
   DATA[797,0] := 2.548442;
   DATA[797,1] := 556.9574;
   DATA[797,2] := 2.0;
   DATA[797,3] := 1.0;
   DATA[797,4] := 262.1764;
   DATA[797,5] := 8.46533;
   DATA[797,6] := 316.2522;
   DATA[797,8] := 1.0;
   DATA[797,9] := 1.0;
   DATA[797,10] := 1.0;
   DATA[797,11] := 2.042384;
   DATA[797,13] := 1010.959;
   DATA[797,14] := 1.0;
   DATA[797,15] := 1.0;
   DATA[797,16] := 1.0;
   DATA[797,17] := 1.0;
   DATA[797,18] := 1.0;
   DATA[797,19] := 1.0;
   DATA[797,20] := 148.808;
   DATA[797,21] := 155.7293;
   DATA[797,22] := 1.717874;
   DATA[797,23] := 978.5183;
   DATA[797,24] := 2.0;
   DATA[797,25] := 2.0;
   DATA[797,26] := 7.878942;
   DATA[797,27] := 144.9116;
   DATA[797,28] := 263.0415;
   DATA[797,29] := 11.95847;
   DATA[797,30] := 1.726352;
   DATA[797,31] := 1.30114;
   DATA[797,32] := 0.7352687;
   DATA[797,33] := 0.3066329;
   DATA[797,34] := 2.0;
   DATA[797,35] := 250.8171;
   DATA[797,36] := 1.69801;
   DATA[797,37] := 189.5828;
   DATA[797,38] := 0.000128152;
   DATA[797,39] := 1.0;
   DATA[798,0] := 2.548442;
   DATA[798,1] := 557.2322;
   DATA[798,2] := 2.0;
   DATA[798,3] := 1.0;
   DATA[798,4] := 262.1764;
   DATA[798,5] := 8.46533;
   DATA[798,6] := 316.2522;
   DATA[798,8] := 1.0;
   DATA[798,9] := 1.0;
   DATA[798,10] := 1.0;
   DATA[798,11] := 2.032781;
   DATA[798,13] := 1011.079;
   DATA[798,14] := 1.0;
   DATA[798,15] := 1.0;
   DATA[798,16] := 1.0;
   DATA[798,17] := 1.0;
   DATA[798,18] := 1.0;
   DATA[798,19] := 1.0;
   DATA[798,20] := 148.808;
   DATA[798,21] := 155.7293;
   DATA[798,22] := 1.717874;
   DATA[798,23] := 978.5183;
   DATA[798,24] := 2.0;
   DATA[798,25] := 2.0;
   DATA[798,26] := 7.878942;
   DATA[798,27] := 144.9116;
   DATA[798,28] := 263.0415;
   DATA[798,29] := 11.95847;
   DATA[798,30] := 1.726352;
   DATA[798,31] := 1.296657;
   DATA[798,32] := 0.7352687;
   DATA[798,33] := 0.3083624;
   DATA[798,34] := 2.0;
   DATA[798,35] := 250.8171;
   DATA[798,36] := 1.69801;
   DATA[798,37] := 189.4867;
   DATA[798,38] := 0.000128152;
   DATA[798,39] := 1.0;
   DATA[799,0] := 2.550684;
   DATA[799,1] := 557.6247;
   DATA[799,2] := 2.0;
   DATA[799,3] := 1.0;
   DATA[799,4] := 262.1764;
   DATA[799,5] := 8.46533;
   DATA[799,6] := 316.2522;
   DATA[799,8] := 1.0;
   DATA[799,9] := 1.0;
   DATA[799,10] := 1.0;
   DATA[799,11] := 2.032781;
   DATA[799,13] := 1010.879;
   DATA[799,14] := 1.0;
   DATA[799,15] := 1.0;
   DATA[799,16] := 1.0;
   DATA[799,17] := 1.0;
   DATA[799,18] := 1.0;
   DATA[799,19] := 1.0;
   DATA[799,20] := 148.808;
   DATA[799,21] := 155.7293;
   DATA[799,22] := 1.717874;
   DATA[799,23] := 977.8646;
   DATA[799,24] := 2.0;
   DATA[799,25] := 2.0;
   DATA[799,26] := 7.878942;
   DATA[799,27] := 144.9116;
   DATA[799,28] := 263.0415;
   DATA[799,29] := 11.95847;
   DATA[799,30] := 1.726352;
   DATA[799,31] := 1.301396;
   DATA[799,32] := 0.7352687;
   DATA[799,33] := 0.3083624;
   DATA[799,34] := 2.0;
   DATA[799,35] := 250.6569;
   DATA[799,36] := 1.69801;
   DATA[799,37] := 189.4867;
   DATA[799,38] := 0.000128152;
   DATA[799,39] := 1.0;
   DATA[800,0] := 2.553246;
   DATA[800,1] := 558.3705;
   DATA[800,2] := 2.0;
   DATA[800,3] := 1.0;
   DATA[800,4] := 262.1764;
   DATA[800,5] := 8.46533;
   DATA[800,6] := 316.2522;
   DATA[800,8] := 1.0;
   DATA[800,9] := 1.0;
   DATA[800,10] := 1.0;
   DATA[800,11] := 2.032781;
   DATA[800,13] := 1011.359;
   DATA[800,14] := 1.0;
   DATA[800,15] := 1.0;
   DATA[800,16] := 1.0;
   DATA[800,17] := 1.0;
   DATA[800,18] := 1.0;
   DATA[800,19] := 1.0;
   DATA[800,20] := 148.808;
   DATA[800,21] := 155.7293;
   DATA[800,22] := 1.717874;
   DATA[800,23] := 977.4417;
   DATA[800,24] := 2.0;
   DATA[800,25] := 2.0;
   DATA[800,26] := 7.878942;
   DATA[800,27] := 144.9116;
   DATA[800,28] := 263.0415;
   DATA[800,29] := 11.95847;
   DATA[800,30] := 1.726352;
   DATA[800,31] := 1.301396;
   DATA[800,32] := 0.7352687;
   DATA[800,33] := 0.3083624;
   DATA[800,34] := 2.0;
   DATA[800,35] := 250.6569;
   DATA[800,36] := 1.69801;
   DATA[800,37] := 189.4867;
   DATA[800,38] := 0.000128152;
   DATA[800,39] := 1.0;
   DATA[801,0] := 2.553246;
   DATA[801,1] := 559.3911;
   DATA[801,2] := 2.0;
   DATA[801,3] := 1.0;
   DATA[801,4] := 262.1764;
   DATA[801,5] := 8.46533;
   DATA[801,6] := 316.0984;
   DATA[801,8] := 1.0;
   DATA[801,9] := 1.0;
   DATA[801,10] := 1.0;
   DATA[801,11] := 2.032781;
   DATA[801,13] := 1011.119;
   DATA[801,14] := 1.0;
   DATA[801,15] := 1.0;
   DATA[801,16] := 1.0;
   DATA[801,17] := 1.0;
   DATA[801,18] := 1.0;
   DATA[801,19] := 1.0;
   DATA[801,20] := 148.808;
   DATA[801,21] := 155.7293;
   DATA[801,22] := 1.717874;
   DATA[801,23] := 976.9034;
   DATA[801,24] := 2.0;
   DATA[801,25] := 2.0;
   DATA[801,26] := 7.878942;
   DATA[801,27] := 144.9116;
   DATA[801,28] := 263.0415;
   DATA[801,29] := 11.95847;
   DATA[801,30] := 1.726352;
   DATA[801,31] := 1.302037;
   DATA[801,32] := 0.7352687;
   DATA[801,33] := 0.3083624;
   DATA[801,34] := 2.0;
   DATA[801,35] := 250.6569;
   DATA[801,36] := 1.69801;
   DATA[801,37] := 189.4867;
   DATA[801,38] := 0.000128152;
   DATA[801,39] := 1.0;
   DATA[802,0] := 2.553246;
   DATA[802,1] := 560.0191;
   DATA[802,2] := 2.0;
   DATA[802,3] := 1.0;
   DATA[802,4] := 262.1764;
   DATA[802,5] := 8.46533;
   DATA[802,6] := 316.0984;
   DATA[802,8] := 1.0;
   DATA[802,9] := 1.0;
   DATA[802,10] := 1.0;
   DATA[802,11] := 2.032781;
   DATA[802,13] := 1011.159;
   DATA[802,14] := 1.0;
   DATA[802,15] := 1.0;
   DATA[802,16] := 1.0;
   DATA[802,17] := 1.0;
   DATA[802,18] := 1.0;
   DATA[802,19] := 1.0;
   DATA[802,20] := 148.808;
   DATA[802,21] := 155.7293;
   DATA[802,22] := 1.717874;
   DATA[802,23] := 976.5573;
   DATA[802,24] := 2.0;
   DATA[802,25] := 2.0;
   DATA[802,26] := 7.878942;
   DATA[802,27] := 144.9116;
   DATA[802,28] := 263.0415;
   DATA[802,29] := 11.95847;
   DATA[802,30] := 1.72725;
   DATA[802,31] := 1.30178;
   DATA[802,32] := 0.7352687;
   DATA[802,33] := 0.3083624;
   DATA[802,34] := 2.0;
   DATA[802,35] := 250.6569;
   DATA[802,36] := 1.69801;
   DATA[802,37] := 189.4867;
   DATA[802,38] := 0.000128152;
   DATA[802,39] := 1.0;
   DATA[803,0] := 2.549082;
   DATA[803,1] := 561.0004;
   DATA[803,2] := 2.0;
   DATA[803,3] := 1.0;
   DATA[803,4] := 262.5288;
   DATA[803,5] := 8.46533;
   DATA[803,6] := 316.0984;
   DATA[803,8] := 1.0;
   DATA[803,9] := 1.0;
   DATA[803,10] := 1.0;
   DATA[803,11] := 2.032781;
   DATA[803,13] := 1010.879;
   DATA[803,14] := 1.0;
   DATA[803,15] := 1.0;
   DATA[803,16] := 1.0;
   DATA[803,17] := 1.0;
   DATA[803,18] := 1.0;
   DATA[803,19] := 1.0;
   DATA[803,20] := 148.808;
   DATA[803,21] := 155.7293;
   DATA[803,22] := 1.717874;
   DATA[803,23] := 976.3651;
   DATA[803,24] := 2.0;
   DATA[803,25] := 2.0;
   DATA[803,26] := 7.878942;
   DATA[803,27] := 145.0141;
   DATA[803,28] := 263.0415;
   DATA[803,29] := 11.95847;
   DATA[803,30] := 1.72725;
   DATA[803,31] := 1.284104;
   DATA[803,32] := 0.7352687;
   DATA[803,33] := 0.3083624;
   DATA[803,34] := 2.0;
   DATA[803,35] := 250.6569;
   DATA[803,36] := 1.778105;
   DATA[803,37] := 189.4867;
   DATA[803,38] := 0.000128152;
   DATA[803,39] := 1.0;
   DATA[804,0] := 2.54652;
   DATA[804,1] := 561.9033;
   DATA[804,2] := 2.0;
   DATA[804,3] := 1.0;
   DATA[804,4] := 262.5288;
   DATA[804,5] := 8.46533;
   DATA[804,6] := 315.9959;
   DATA[804,8] := 1.0;
   DATA[804,9] := 1.0;
   DATA[804,10] := 1.0;
   DATA[804,11] := 2.032781;
   DATA[804,13] := 1010.879;
   DATA[804,14] := 1.0;
   DATA[804,15] := 1.0;
   DATA[804,16] := 1.0;
   DATA[804,17] := 1.0;
   DATA[804,18] := 1.0;
   DATA[804,19] := 1.0;
   DATA[804,20] := 148.808;
   DATA[804,21] := 155.7293;
   DATA[804,22] := 1.717874;
   DATA[804,23] := 976.1728;
   DATA[804,24] := 2.0;
   DATA[804,25] := 2.0;
   DATA[804,26] := 7.878942;
   DATA[804,27] := 145.0141;
   DATA[804,28] := 263.0415;
   DATA[804,29] := 12.03538;
   DATA[804,30] := 1.72725;
   DATA[804,31] := 1.267709;
   DATA[804,32] := 0.7352687;
   DATA[804,33] := 0.3080421;
   DATA[804,34] := 2.0;
   DATA[804,35] := 250.737;
   DATA[804,36] := 1.778105;
   DATA[804,37] := 189.4867;
   DATA[804,38] := 0.000128152;
   DATA[804,39] := 1.0;
   DATA[805,0] := 2.54652;
   DATA[805,1] := 562.8845;
   DATA[805,2] := 2.0;
   DATA[805,3] := 1.0;
   DATA[805,4] := 262.5288;
   DATA[805,5] := 8.46533;
   DATA[805,6] := 315.8677;
   DATA[805,8] := 1.0;
   DATA[805,9] := 1.0;
   DATA[805,10] := 1.0;
   DATA[805,11] := 2.032781;
   DATA[805,13] := 1011.079;
   DATA[805,14] := 1.0;
   DATA[805,15] := 1.0;
   DATA[805,16] := 1.0;
   DATA[805,17] := 1.0;
   DATA[805,18] := 1.0;
   DATA[805,19] := 1.0;
   DATA[805,20] := 148.808;
   DATA[805,21] := 155.7293;
   DATA[805,22] := 1.717874;
   DATA[805,23] := 975.9421;
   DATA[805,24] := 2.0;
   DATA[805,25] := 2.0;
   DATA[805,26] := 7.878942;
   DATA[805,27] := 145.0141;
   DATA[805,28] := 263.0415;
   DATA[805,29] := 12.22763;
   DATA[805,30] := 1.72725;
   DATA[805,31] := 1.261688;
   DATA[805,32] := 0.7352687;
   DATA[805,33] := 0.3069532;
   DATA[805,34] := 2.0;
   DATA[805,35] := 250.785;
   DATA[805,36] := 1.778105;
   DATA[805,37] := 189.4867;
   DATA[805,38] := 0.000128152;
   DATA[805,39] := 1.0;
   DATA[806,0] := 2.54652;
   DATA[806,1] := 563.9052;
   DATA[806,2] := 2.0;
   DATA[806,3] := 1.0;
   DATA[806,4] := 262.2404;
   DATA[806,5] := 8.46533;
   DATA[806,6] := 315.8677;
   DATA[806,8] := 1.0;
   DATA[806,9] := 1.0;
   DATA[806,10] := 1.0;
   DATA[806,11] := 2.032781;
   DATA[806,13] := 1011.119;
   DATA[806,14] := 1.0;
   DATA[806,15] := 1.0;
   DATA[806,16] := 1.0;
   DATA[806,17] := 1.0;
   DATA[806,18] := 1.0;
   DATA[806,19] := 1.0;
   DATA[806,20] := 148.808;
   DATA[806,21] := 155.7293;
   DATA[806,22] := 1.717874;
   DATA[806,23] := 975.596;
   DATA[806,24] := 2.0;
   DATA[806,25] := 2.0;
   DATA[806,26] := 7.878942;
   DATA[806,27] := 145.0141;
   DATA[806,28] := 263.0415;
   DATA[806,29] := 12.22763;
   DATA[806,30] := 1.72725;
   DATA[806,31] := 1.255284;
   DATA[806,32] := 0.7352687;
   DATA[806,33] := 0.3069532;
   DATA[806,34] := 2.0;
   DATA[806,35] := 250.785;
   DATA[806,36] := 1.778105;
   DATA[806,37] := 189.4867;
   DATA[806,38] := 0.000128152;
   DATA[806,39] := 1.0;
   DATA[807,0] := 2.540115;
   DATA[807,1] := 564.8079;
   DATA[807,2] := 2.0;
   DATA[807,3] := 1.0;
   DATA[807,4] := 262.2404;
   DATA[807,5] := 8.46533;
   DATA[807,6] := 315.7396;
   DATA[807,8] := 1.0;
   DATA[807,9] := 1.0;
   DATA[807,10] := 1.0;
   DATA[807,11] := 2.032781;
   DATA[807,13] := 1011.359;
   DATA[807,14] := 1.0;
   DATA[807,15] := 1.0;
   DATA[807,16] := 1.0;
   DATA[807,17] := 1.0;
   DATA[807,18] := 1.0;
   DATA[807,19] := 1.0;
   DATA[807,20] := 148.808;
   DATA[807,21] := 155.7293;
   DATA[807,22] := 1.717874;
   DATA[807,23] := 975.0192;
   DATA[807,24] := 2.0;
   DATA[807,25] := 2.0;
   DATA[807,26] := 7.878942;
   DATA[807,27] := 145.0141;
   DATA[807,28] := 263.0415;
   DATA[807,29] := 12.22763;
   DATA[807,30] := 1.72725;
   DATA[807,31] := 1.254771;
   DATA[807,32] := 0.7352687;
   DATA[807,33] := 0.3081703;
   DATA[807,34] := 2.0;
   DATA[807,35] := 250.785;
   DATA[807,36] := 1.778105;
   DATA[807,37] := 189.4867;
   DATA[807,38] := 0.000128152;
   DATA[807,39] := 1.0;
   DATA[808,0] := 2.540115;
   DATA[808,1] := 565.2004;
   DATA[808,2] := 2.0;
   DATA[808,3] := 1.0;
   DATA[808,4] := 262.2404;
   DATA[808,5] := 8.46533;
   DATA[808,6] := 315.5858;
   DATA[808,8] := 1.0;
   DATA[808,9] := 1.0;
   DATA[808,10] := 1.0;
   DATA[808,11] := 2.032781;
   DATA[808,13] := 1010.919;
   DATA[808,14] := 1.0;
   DATA[808,15] := 1.0;
   DATA[808,16] := 1.0;
   DATA[808,17] := 1.0;
   DATA[808,18] := 1.0;
   DATA[808,19] := 1.0;
   DATA[808,20] := 148.808;
   DATA[808,21] := 155.7293;
   DATA[808,22] := 1.717874;
   DATA[808,23] := 974.6732;
   DATA[808,24] := 2.0;
   DATA[808,25] := 2.0;
   DATA[808,26] := 7.878942;
   DATA[808,27] := 145.0141;
   DATA[808,28] := 263.0415;
   DATA[808,29] := 12.22763;
   DATA[808,30] := 1.729172;
   DATA[808,31] := 1.270142;
   DATA[808,32] := 0.7352687;
   DATA[808,33] := 0.3081703;
   DATA[808,34] := 2.0;
   DATA[808,35] := 250.6729;
   DATA[808,36] := 1.649953;
   DATA[808,37] := 189.4867;
   DATA[808,38] := 0.000128152;
   DATA[808,39] := 1.0;
   DATA[809,0] := 2.551645;
   DATA[809,1] := 565.3967;
   DATA[809,2] := 2.0;
   DATA[809,3] := 1.0;
   DATA[809,4] := 262.2404;
   DATA[809,5] := 8.46533;
   DATA[809,6] := 315.5858;
   DATA[809,8] := 1.0;
   DATA[809,9] := 1.0;
   DATA[809,10] := 1.0;
   DATA[809,11] := 2.032781;
   DATA[809,13] := 1010.959;
   DATA[809,14] := 1.0;
   DATA[809,15] := 1.0;
   DATA[809,16] := 1.0;
   DATA[809,17] := 1.0;
   DATA[809,18] := 1.0;
   DATA[809,19] := 1.0;
   DATA[809,20] := 148.808;
   DATA[809,21] := 155.7293;
   DATA[809,22] := 1.717874;
   DATA[809,23] := 974.6347;
   DATA[809,24] := 2.0;
   DATA[809,25] := 2.0;
   DATA[809,26] := 7.878942;
   DATA[809,27] := 144.7578;
   DATA[809,28] := 263.0415;
   DATA[809,29] := 12.22763;
   DATA[809,30] := 1.729172;
   DATA[809,31] := 1.272576;
   DATA[809,32] := 0.7352687;
   DATA[809,33] := 0.3083624;
   DATA[809,34] := 2.0;
   DATA[809,35] := 250.5608;
   DATA[809,36] := 1.649953;
   DATA[809,37] := 189.3425;
   DATA[809,38] := 0.000128152;
   DATA[809,39] := 1.0;
   DATA[810,0] := 2.553886;
   DATA[810,1] := 565.5145;
   DATA[810,2] := 2.0;
   DATA[810,3] := 1.0;
   DATA[810,4] := 262.2404;
   DATA[810,5] := 8.46533;
   DATA[810,6] := 315.5601;
   DATA[810,8] := 1.0;
   DATA[810,9] := 1.0;
   DATA[810,10] := 1.0;
   DATA[810,11] := 2.032781;
   DATA[810,13] := 1011.039;
   DATA[810,14] := 1.0;
   DATA[810,15] := 1.0;
   DATA[810,16] := 1.0;
   DATA[810,17] := 1.0;
   DATA[810,18] := 1.0;
   DATA[810,19] := 1.0;
   DATA[810,20] := 148.808;
   DATA[810,21] := 155.7293;
   DATA[810,22] := 1.716849;
   DATA[810,23] := 974.1733;
   DATA[810,24] := 2.0;
   DATA[810,25] := 2.0;
   DATA[810,26] := 7.878942;
   DATA[810,27] := 144.7578;
   DATA[810,28] := 263.0415;
   DATA[810,29] := 12.22763;
   DATA[810,30] := 1.7293;
   DATA[810,31] := 1.272576;
   DATA[810,32] := 0.7352687;
   DATA[810,33] := 0.3072735;
   DATA[810,34] := 2.0;
   DATA[810,35] := 250.5608;
   DATA[810,36] := 1.649953;
   DATA[810,37] := 189.3425;
   DATA[810,38] := 0.000128152;
   DATA[810,39] := 1.0;
   DATA[811,0] := 2.554527;
   DATA[811,1] := 565.279;
   DATA[811,2] := 2.0;
   DATA[811,3] := 1.0;
   DATA[811,4] := 262.2404;
   DATA[811,5] := 8.46533;
   DATA[811,6] := 315.5601;
   DATA[811,8] := 1.0;
   DATA[811,9] := 1.0;
   DATA[811,10] := 1.0;
   DATA[811,11] := 2.032781;
   DATA[811,13] := 1010.718;
   DATA[811,14] := 1.0;
   DATA[811,15] := 1.0;
   DATA[811,16] := 1.0;
   DATA[811,17] := 1.0;
   DATA[811,18] := 1.0;
   DATA[811,19] := 1.0;
   DATA[811,20] := 148.808;
   DATA[811,21] := 155.7293;
   DATA[811,22] := 1.71608;
   DATA[811,23] := 973.7888;
   DATA[811,24] := 2.0;
   DATA[811,25] := 2.0;
   DATA[811,26] := 7.878942;
   DATA[811,27] := 144.7578;
   DATA[811,28] := 263.0415;
   DATA[811,29] := 11.84312;
   DATA[811,30] := 1.7293;
   DATA[811,31] := 1.272192;
   DATA[811,32] := 0.7352687;
   DATA[811,33] := 0.3068251;
   DATA[811,34] := 2.0;
   DATA[811,35] := 250.5608;
   DATA[811,36] := 1.649953;
   DATA[811,37] := 189.3425;
   DATA[811,38] := 0.000128152;
   DATA[811,39] := 1.0;
   DATA[812,0] := 2.554527;
   DATA[812,1] := 565.2397;
   DATA[812,2] := 2.0;
   DATA[812,3] := 1.0;
   DATA[812,4] := 262.2404;
   DATA[812,5] := 8.46533;
   DATA[812,6] := 315.5601;
   DATA[812,8] := 1.0;
   DATA[812,9] := 1.0;
   DATA[812,10] := 1.0;
   DATA[812,11] := 2.032781;
   DATA[812,13] := 1010.278;
   DATA[812,14] := 1.0;
   DATA[812,15] := 1.0;
   DATA[812,16] := 1.0;
   DATA[812,17] := 1.0;
   DATA[812,18] := 1.0;
   DATA[812,19] := 1.0;
   DATA[812,20] := 148.808;
   DATA[812,21] := 155.7293;
   DATA[812,22] := 1.715567;
   DATA[812,23] := 973.2889;
   DATA[812,24] := 2.0;
   DATA[812,25] := 2.0;
   DATA[812,26] := 7.878942;
   DATA[812,27] := 144.7578;
   DATA[812,28] := 263.0415;
   DATA[812,29] := 11.84312;
   DATA[812,30] := 1.7293;
   DATA[812,31] := 1.272576;
   DATA[812,32] := 0.7352687;
   DATA[812,33] := 0.3083624;
   DATA[812,34] := 2.0;
   DATA[812,35] := 250.5608;
   DATA[812,36] := 1.649953;
   DATA[812,37] := 189.3425;
   DATA[812,38] := 0.000128152;
   DATA[812,39] := 1.0;
   DATA[813,0] := 2.554527;
   DATA[813,1] := 565.3182;
   DATA[813,2] := 2.0;
   DATA[813,3] := 1.0;
   DATA[813,4] := 262.2404;
   DATA[813,5] := 8.46533;
   DATA[813,6] := 315.5601;
   DATA[813,8] := 1.0;
   DATA[813,9] := 1.0;
   DATA[813,10] := 1.0;
   DATA[813,11] := 2.032781;
   DATA[813,13] := 1010.758;
   DATA[813,14] := 1.0;
   DATA[813,15] := 1.0;
   DATA[813,16] := 1.0;
   DATA[813,17] := 1.0;
   DATA[813,18] := 1.0;
   DATA[813,19] := 1.0;
   DATA[813,20] := 148.808;
   DATA[813,21] := 155.7293;
   DATA[813,22] := 1.715439;
   DATA[813,23] := 972.5198;
   DATA[813,24] := 2.0;
   DATA[813,25] := 2.0;
   DATA[813,26] := 7.878942;
   DATA[813,27] := 144.7578;
   DATA[813,28] := 263.0415;
   DATA[813,29] := 11.84312;
   DATA[813,30] := 1.726993;
   DATA[813,31] := 1.289996;
   DATA[813,32] := 0.7352687;
   DATA[813,33] := 0.3083624;
   DATA[813,34] := 2.0;
   DATA[813,35] := 250.5608;
   DATA[813,36] := 1.746067;
   DATA[813,37] := 189.3425;
   DATA[813,38] := 0.000128152;
   DATA[813,39] := 1.0;
   DATA[814,0] := 2.55837;
   DATA[814,1] := 565.2004;
   DATA[814,2] := 2.0;
   DATA[814,3] := 1.0;
   DATA[814,4] := 262.2404;
   DATA[814,5] := 8.46533;
   DATA[814,6] := 315.3807;
   DATA[814,8] := 1.0;
   DATA[814,9] := 1.0;
   DATA[814,10] := 1.0;
   DATA[814,11] := 2.032781;
   DATA[814,13] := 1010.478;
   DATA[814,14] := 1.0;
   DATA[814,15] := 1.0;
   DATA[814,16] := 1.0;
   DATA[814,17] := 1.0;
   DATA[814,18] := 1.0;
   DATA[814,19] := 1.0;
   DATA[814,20] := 148.808;
   DATA[814,21] := 155.7293;
   DATA[814,22] := 1.715439;
   DATA[814,23] := 972.2507;
   DATA[814,24] := 2.0;
   DATA[814,25] := 2.0;
   DATA[814,26] := 7.878942;
   DATA[814,27] := 144.7578;
   DATA[814,28] := 263.0415;
   DATA[814,29] := 12.11228;
   DATA[814,30] := 1.726993;
   DATA[814,31] := 1.30178;
   DATA[814,32] := 0.7352687;
   DATA[814,33] := 0.3083624;
   DATA[814,34] := 2.0;
   DATA[814,35] := 250.5608;
   DATA[814,36] := 1.746067;
   DATA[814,37] := 189.3425;
   DATA[814,38] := 0.000128152;
   DATA[814,39] := 1.0;
   DATA[815,0] := 2.55837;
   DATA[815,1] := 564.8079;
   DATA[815,2] := 2.0;
   DATA[815,3] := 1.0;
   DATA[815,4] := 262.2404;
   DATA[815,5] := 8.46533;
   DATA[815,6] := 315.3807;
   DATA[815,8] := 1.0;
   DATA[815,9] := 1.0;
   DATA[815,10] := 1.0;
   DATA[815,11] := 2.032781;
   DATA[815,13] := 1010.638;
   DATA[815,14] := 1.0;
   DATA[815,15] := 1.0;
   DATA[815,16] := 1.0;
   DATA[815,17] := 1.0;
   DATA[815,18] := 1.0;
   DATA[815,19] := 1.0;
   DATA[815,20] := 148.808;
   DATA[815,21] := 155.7293;
   DATA[815,22] := 1.715439;
   DATA[815,23] := 972.1354;
   DATA[815,24] := 2.0;
   DATA[815,25] := 2.0;
   DATA[815,26] := 7.878942;
   DATA[815,27] := 144.7578;
   DATA[815,28] := 263.0415;
   DATA[815,29] := 12.11228;
   DATA[815,30] := 1.726993;
   DATA[815,31] := 1.30178;
   DATA[815,32] := 0.7352687;
   DATA[815,33] := 0.3083624;
   DATA[815,34] := 2.0;
   DATA[815,35] := 250.5608;
   DATA[815,36] := 1.746067;
   DATA[815,37] := 189.3425;
   DATA[815,38] := 0.000128152;
   DATA[815,39] := 1.0;
   DATA[816,0] := 2.55837;
   DATA[816,1] := 564.8472;
   DATA[816,2] := 2.0;
   DATA[816,3] := 1.0;
   DATA[816,4] := 262.2404;
   DATA[816,5] := 8.46533;
   DATA[816,6] := 315.3807;
   DATA[816,8] := 1.0;
   DATA[816,9] := 1.0;
   DATA[816,10] := 1.0;
   DATA[816,11] := 2.032781;
   DATA[816,13] := 1010.478;
   DATA[816,14] := 1.0;
   DATA[816,15] := 1.0;
   DATA[816,16] := 1.0;
   DATA[816,17] := 1.0;
   DATA[816,18] := 1.0;
   DATA[816,19] := 1.0;
   DATA[816,20] := 148.808;
   DATA[816,21] := 155.7293;
   DATA[816,22] := 1.715439;
   DATA[816,23] := 971.8662;
   DATA[816,24] := 2.0;
   DATA[816,25] := 2.0;
   DATA[816,26] := 7.878942;
   DATA[816,27] := 144.7578;
   DATA[816,28] := 263.0415;
   DATA[816,29] := 12.11228;
   DATA[816,30] := 1.726993;
   DATA[816,31] := 1.296401;
   DATA[816,32] := 0.7352687;
   DATA[816,33] := 0.3083624;
   DATA[816,34] := 2.0;
   DATA[816,35] := 250.5608;
   DATA[816,36] := 1.746067;
   DATA[816,37] := 189.3425;
   DATA[816,38] := 0.000128152;
   DATA[816,39] := 1.0;
   DATA[817,0] := 2.557089;
   DATA[817,1] := 564.6509;
   DATA[817,2] := 2.0;
   DATA[817,3] := 1.0;
   DATA[817,4] := 262.2404;
   DATA[817,5] := 8.46533;
   DATA[817,6] := 315.3807;
   DATA[817,8] := 1.0;
   DATA[817,9] := 1.0;
   DATA[817,10] := 1.0;
   DATA[817,11] := 2.032781;
   DATA[817,13] := 1010.638;
   DATA[817,14] := 1.0;
   DATA[817,15] := 1.0;
   DATA[817,16] := 1.0;
   DATA[817,17] := 1.0;
   DATA[817,18] := 1.0;
   DATA[817,19] := 1.0;
   DATA[817,20] := 148.808;
   DATA[817,21] := 155.7293;
   DATA[817,22] := 1.716721;
   DATA[817,23] := 971.4432;
   DATA[817,24] := 2.0;
   DATA[817,25] := 2.0;
   DATA[817,26] := 7.878942;
   DATA[817,27] := 144.7578;
   DATA[817,28] := 263.0415;
   DATA[817,29] := 12.11228;
   DATA[817,30] := 1.72507;
   DATA[817,31] := 1.291149;
   DATA[817,32] := 0.7352687;
   DATA[817,33] := 0.3083624;
   DATA[817,34] := 2.0;
   DATA[817,35] := 250.5608;
   DATA[817,36] := 1.746067;
   DATA[817,37] := 189.3425;
   DATA[817,38] := 0.000128152;
   DATA[817,39] := 1.0;
   DATA[818,0] := 2.548121;
   DATA[818,1] := 564.4547;
   DATA[818,2] := 2.0;
   DATA[818,3] := 1.0;
   DATA[818,4] := 262.2404;
   DATA[818,5] := 8.46533;
   DATA[818,6] := 315.3807;
   DATA[818,8] := 1.0;
   DATA[818,9] := 1.0;
   DATA[818,10] := 1.0;
   DATA[818,11] := 2.032781;
   DATA[818,13] := 1010.438;
   DATA[818,14] := 1.0;
   DATA[818,15] := 1.0;
   DATA[818,16] := 1.0;
   DATA[818,17] := 1.0;
   DATA[818,18] := 1.0;
   DATA[818,19] := 1.0;
   DATA[818,20] := 148.808;
   DATA[818,21] := 155.7293;
   DATA[818,22] := 1.717489;
   DATA[818,23] := 971.2894;
   DATA[818,24] := 2.0;
   DATA[818,25] := 2.0;
   DATA[818,26] := 7.878942;
   DATA[818,27] := 144.7578;
   DATA[818,28] := 263.0415;
   DATA[818,29] := 12.11228;
   DATA[818,30] := 1.72507;
   DATA[818,31] := 1.291149;
   DATA[818,32] := 0.7352687;
   DATA[818,33] := 0.3083624;
   DATA[818,34] := 2.0;
   DATA[818,35] := 250.5608;
   DATA[818,36] := 1.746067;
   DATA[818,37] := 189.3425;
   DATA[818,38] := 0.000128152;
   DATA[818,39] := 1.0;
   DATA[819,0] := 2.548121;
   DATA[819,1] := 565.2004;
   DATA[819,2] := 2.0;
   DATA[819,3] := 1.0;
   DATA[819,4] := 262.2404;
   DATA[819,5] := 8.46533;
   DATA[819,6] := 315.3807;
   DATA[819,8] := 1.0;
   DATA[819,9] := 1.0;
   DATA[819,10] := 1.0;
   DATA[819,11] := 2.032781;
   DATA[819,13] := 1010.558;
   DATA[819,14] := 1.0;
   DATA[819,15] := 1.0;
   DATA[819,16] := 1.0;
   DATA[819,17] := 1.0;
   DATA[819,18] := 1.0;
   DATA[819,19] := 1.0;
   DATA[819,20] := 148.808;
   DATA[819,21] := 155.7293;
   DATA[819,22] := 1.717489;
   DATA[819,23] := 970.7896;
   DATA[819,24] := 2.0;
   DATA[819,25] := 2.0;
   DATA[819,26] := 7.878942;
   DATA[819,27] := 144.7578;
   DATA[819,28] := 263.0415;
   DATA[819,29] := 12.11228;
   DATA[819,30] := 1.72507;
   DATA[819,31] := 1.291149;
   DATA[819,32] := 0.7352687;
   DATA[819,33] := 0.3083624;
   DATA[819,34] := 2.0;
   DATA[819,35] := 250.5608;
   DATA[819,36] := 1.746067;
   DATA[819,37] := 189.3425;
   DATA[819,38] := 0.000128152;
   DATA[819,39] := 1.0;
   DATA[820,0] := 2.543638;
   DATA[820,1] := 565.593;
   DATA[820,2] := 2.0;
   DATA[820,3] := 1.0;
   DATA[820,4] := 262.3366;
   DATA[820,5] := 8.46533;
   DATA[820,6] := 315.3807;
   DATA[820,8] := 1.0;
   DATA[820,9] := 1.0;
   DATA[820,10] := 1.0;
   DATA[820,11] := 2.032781;
   DATA[820,13] := 1010.438;
   DATA[820,14] := 1.0;
   DATA[820,15] := 1.0;
   DATA[820,16] := 1.0;
   DATA[820,17] := 1.0;
   DATA[820,18] := 1.0;
   DATA[820,19] := 1.0;
   DATA[820,20] := 148.808;
   DATA[820,21] := 155.7293;
   DATA[820,22] := 1.717489;
   DATA[820,23] := 970.5973;
   DATA[820,24] := 2.0;
   DATA[820,25] := 2.0;
   DATA[820,26] := 7.878942;
   DATA[820,27] := 144.7578;
   DATA[820,28] := 263.0415;
   DATA[820,29] := 12.11228;
   DATA[820,30] := 1.72507;
   DATA[820,31] := 1.291149;
   DATA[820,32] := 0.7352687;
   DATA[820,33] := 0.3083624;
   DATA[820,34] := 2.0;
   DATA[820,35] := 250.5608;
   DATA[820,36] := 1.730048;
   DATA[820,37] := 189.3425;
   DATA[820,38] := 0.000128152;
   DATA[820,39] := 1.0;
   DATA[821,0] := 2.543638;
   DATA[821,1] := 566.7706;
   DATA[821,2] := 2.0;
   DATA[821,3] := 1.0;
   DATA[821,4] := 262.3366;
   DATA[821,5] := 8.46533;
   DATA[821,6] := 315.3807;
   DATA[821,8] := 1.0;
   DATA[821,9] := 1.0;
   DATA[821,10] := 1.0;
   DATA[821,11] := 2.032781;
   DATA[821,13] := 1010.078;
   DATA[821,14] := 1.0;
   DATA[821,15] := 1.0;
   DATA[821,16] := 1.0;
   DATA[821,17] := 1.0;
   DATA[821,18] := 1.0;
   DATA[821,19] := 1.0;
   DATA[821,20] := 148.808;
   DATA[821,21] := 155.7037;
   DATA[821,22] := 1.717489;
   DATA[821,23] := 970.3666;
   DATA[821,24] := 2.0;
   DATA[821,25] := 2.0;
   DATA[821,26] := 7.878942;
   DATA[821,27] := 144.7578;
   DATA[821,28] := 263.0415;
   DATA[821,29] := 12.11228;
   DATA[821,30] := 1.72507;
   DATA[821,31] := 1.301652;
   DATA[821,32] := 0.7352687;
   DATA[821,33] := 0.3083624;
   DATA[821,34] := 2.0;
   DATA[821,35] := 250.5608;
   DATA[821,36] := 1.730048;
   DATA[821,37] := 189.3425;
   DATA[821,38] := 0.000128152;
   DATA[821,39] := 1.0;
   DATA[822,0] := 2.543638;
   DATA[822,1] := 567.3594;
   DATA[822,2] := 2.0;
   DATA[822,3] := 1.0;
   DATA[822,4] := 262.3366;
   DATA[822,5] := 8.46533;
   DATA[822,6] := 315.1243;
   DATA[822,8] := 1.0;
   DATA[822,9] := 1.0;
   DATA[822,10] := 1.0;
   DATA[822,11] := 2.032781;
   DATA[822,13] := 1010.118;
   DATA[822,14] := 1.0;
   DATA[822,15] := 1.0;
   DATA[822,16] := 1.0;
   DATA[822,17] := 1.0;
   DATA[822,18] := 1.0;
   DATA[822,19] := 1.0;
   DATA[822,20] := 148.808;
   DATA[822,21] := 155.6011;
   DATA[822,22] := 1.717489;
   DATA[822,23] := 970.1359;
   DATA[822,24] := 2.0;
   DATA[822,25] := 2.0;
   DATA[822,26] := 7.878942;
   DATA[822,27] := 144.7578;
   DATA[822,28] := 263.0415;
   DATA[822,29] := 12.11228;
   DATA[822,30] := 1.72507;
   DATA[822,31] := 1.29845;
   DATA[822,32] := 0.7352687;
   DATA[822,33] := 0.3083624;
   DATA[822,34] := 2.0;
   DATA[822,35] := 250.5608;
   DATA[822,36] := 1.730048;
   DATA[822,37] := 189.4066;
   DATA[822,38] := 0.000128152;
   DATA[822,39] := 1.0;
   DATA[823,0] := 2.542677;
   DATA[823,1] := 567.7911;
   DATA[823,2] := 2.0;
   DATA[823,3] := 1.0;
   DATA[823,4] := 262.3366;
   DATA[823,5] := 8.46533;
   DATA[823,6] := 315.1243;
   DATA[823,8] := 1.0;
   DATA[823,9] := 1.0;
   DATA[823,10] := 1.0;
   DATA[823,11] := 2.032781;
   DATA[823,13] := 1010.118;
   DATA[823,14] := 1.0;
   DATA[823,15] := 1.0;
   DATA[823,16] := 1.0;
